  PROC DrawPart130()
    MoveL Offs(pOrigin,337.86,23.80,0.00),v40,fine,tPen\WObj:=wPaper;
    MoveL Offs(pOrigin,337.86,23.80,6.00),v60,z5,tPen\WObj:=wPaper;
    MoveL Offs(pOrigin,338.99,27.95,6.00),vTravel,z5,tPen\WObj:=wPaper;
    MoveL Offs(pOrigin,338.99,27.95,0.00),v60,z0,tPen\WObj:=wPaper;
    MoveL Offs(pOrigin,338.99,29.01,0.00),v40,fine,tPen\WObj:=wPaper;
    MoveL Offs(pOrigin,338.99,29.01,6.00),v60,z5,tPen\WObj:=wPaper;
    MoveL Offs(pOrigin,338.73,31.88,6.00),vTravel,z5,tPen\WObj:=wPaper;
    MoveL Offs(pOrigin,338.73,31.88,0.00),v60,z0,tPen\WObj:=wPaper;
    MoveL Offs(pOrigin,336.63,33.99,0.00),v40,fine,tPen\WObj:=wPaper;
    MoveL Offs(pOrigin,336.63,33.99,6.00),v60,z5,tPen\WObj:=wPaper;
    MoveL Offs(pOrigin,334.79,36.45,6.00),vTravel,z5,tPen\WObj:=wPaper;
    MoveL Offs(pOrigin,334.79,36.45,0.00),v60,z0,tPen\WObj:=wPaper;
    MoveL Offs(pOrigin,334.36,34.11,0.00),v40,z0,tPen\WObj:=wPaper;
    MoveL Offs(pOrigin,334.36,32.62,0.00),v40,z0,tPen\WObj:=wPaper;
    MoveL Offs(pOrigin,334.79,31.14,0.00),v40,fine,tPen\WObj:=wPaper;
    MoveL Offs(pOrigin,334.79,31.14,6.00),v60,z5,tPen\WObj:=wPaper;
    MoveL Offs(pOrigin,330.05,28.61,6.00),vTravel,z5,tPen\WObj:=wPaper;
    MoveL Offs(pOrigin,330.05,28.61,0.00),v60,z0,tPen\WObj:=wPaper;
    MoveL Offs(pOrigin,332.76,25.91,0.00),v40,fine,tPen\WObj:=wPaper;
    MoveL Offs(pOrigin,332.76,25.91,6.00),v60,z5,tPen\WObj:=wPaper;
    MoveL Offs(pOrigin,324.97,24.73,6.00),vTravel,z5,tPen\WObj:=wPaper;
    MoveL Offs(pOrigin,324.97,24.73,0.00),v60,z0,tPen\WObj:=wPaper;
    MoveL Offs(pOrigin,317.76,31.95,0.00),v40,z0,tPen\WObj:=wPaper;
    MoveL Offs(pOrigin,318.38,31.94,0.00),v40,z0,tPen\WObj:=wPaper;
    MoveL Offs(pOrigin,312.97,26.53,0.00),v40,z0,tPen\WObj:=wPaper;
    MoveL Offs(pOrigin,313.75,26.62,0.00),v40,z0,tPen\WObj:=wPaper;
    MoveL Offs(pOrigin,319.49,26.62,0.00),v40,fine,tPen\WObj:=wPaper;
    MoveL Offs(pOrigin,319.49,26.62,6.00),v60,z5,tPen\WObj:=wPaper;
    MoveL Offs(pOrigin,320.12,27.67,6.00),vTravel,z5,tPen\WObj:=wPaper;
    MoveL Offs(pOrigin,320.12,27.67,0.00),v60,z0,tPen\WObj:=wPaper;
    MoveL Offs(pOrigin,310.99,27.67,0.00),v40,z0,tPen\WObj:=wPaper;
    MoveL Offs(pOrigin,310.58,28.67,0.00),v40,z0,tPen\WObj:=wPaper;
    MoveL Offs(pOrigin,314.04,25.22,0.00),v40,z0,tPen\WObj:=wPaper;
    MoveL Offs(pOrigin,314.02,26.08,0.00),v40,z0,tPen\WObj:=wPaper;
    MoveL Offs(pOrigin,324.54,36.60,0.00),v40,z0,tPen\WObj:=wPaper;
    MoveL Offs(pOrigin,325.24,36.42,0.00),v40,z0,tPen\WObj:=wPaper;
    MoveL Offs(pOrigin,321.93,39.72,0.00),v40,z0,tPen\WObj:=wPaper;
    MoveL Offs(pOrigin,322.75,39.29,0.00),v40,z0,tPen\WObj:=wPaper;
    MoveL Offs(pOrigin,324.85,41.40,0.00),v40,z0,tPen\WObj:=wPaper;
    MoveL Offs(pOrigin,325.67,41.96,0.00),v40,z0,tPen\WObj:=wPaper;
    MoveL Offs(pOrigin,321.31,46.32,0.00),v40,z0,tPen\WObj:=wPaper;
    MoveL Offs(pOrigin,322.17,46.18,0.00),v40,z0,tPen\WObj:=wPaper;
    MoveL Offs(pOrigin,324.27,48.29,0.00),v40,fine,tPen\WObj:=wPaper;
    MoveL Offs(pOrigin,324.27,48.29,6.00),v60,z5,tPen\WObj:=wPaper;
    MoveL Offs(pOrigin,324.57,47.09,6.00),vTravel,z5,tPen\WObj:=wPaper;
    MoveL Offs(pOrigin,324.57,47.09,0.00),v60,z0,tPen\WObj:=wPaper;
    MoveL Offs(pOrigin,322.47,44.98,0.00),v40,z0,tPen\WObj:=wPaper;
    MoveL Offs(pOrigin,323.10,45.62,0.00),v40,z0,tPen\WObj:=wPaper;
    MoveL Offs(pOrigin,324.16,45.62,0.00),v40,z0,tPen\WObj:=wPaper;
    MoveL Offs(pOrigin,324.72,45.74,0.00),v40,z0,tPen\WObj:=wPaper;
    MoveL Offs(pOrigin,322.76,43.79,0.00),v40,z0,tPen\WObj:=wPaper;
    MoveL Offs(pOrigin,321.77,44.37,0.00),v40,z0,tPen\WObj:=wPaper;
    MoveL Offs(pOrigin,325.67,40.46,0.00),v40,z0,tPen\WObj:=wPaper;
    MoveL Offs(pOrigin,324.85,39.90,0.00),v40,z0,tPen\WObj:=wPaper;
    MoveL Offs(pOrigin,322.29,37.34,0.00),v40,z0,tPen\WObj:=wPaper;
    MoveL Offs(pOrigin,321.79,36.88,0.00),v40,z0,tPen\WObj:=wPaper;
    MoveL Offs(pOrigin,324.65,34.02,0.00),v40,z0,tPen\WObj:=wPaper;
    MoveL Offs(pOrigin,324.08,34.65,0.00),v40,z0,tPen\WObj:=wPaper;
    MoveL Offs(pOrigin,315.22,25.79,0.00),v40,z0,tPen\WObj:=wPaper;
    MoveL Offs(pOrigin,316.26,25.34,0.00),v40,z0,tPen\WObj:=wPaper;
    MoveL Offs(pOrigin,323.78,32.85,0.00),v40,z0,tPen\WObj:=wPaper;
    MoveL Offs(pOrigin,323.31,32.95,0.00),v40,z0,tPen\WObj:=wPaper;
    MoveL Offs(pOrigin,321.19,32.95,0.00),v40,z0,tPen\WObj:=wPaper;
    MoveL Offs(pOrigin,321.04,32.41,0.00),v40,z0,tPen\WObj:=wPaper;
    MoveL Offs(pOrigin,321.04,31.14,0.00),v40,z0,tPen\WObj:=wPaper;
    MoveL Offs(pOrigin,322.09,31.56,0.00),v40,z0,tPen\WObj:=wPaper;
    MoveL Offs(pOrigin,322.09,33.69,0.00),v40,z0,tPen\WObj:=wPaper;
    MoveL Offs(pOrigin,322.04,34.01,0.00),v40,z0,tPen\WObj:=wPaper;
    MoveL Offs(pOrigin,323.52,34.01,0.00),v40,z0,tPen\WObj:=wPaper;
    MoveL Offs(pOrigin,323.74,35.06,0.00),v40,z0,tPen\WObj:=wPaper;
    MoveL Offs(pOrigin,322.46,35.06,0.00),v40,z0,tPen\WObj:=wPaper;
    MoveL Offs(pOrigin,321.39,34.94,0.00),v40,z0,tPen\WObj:=wPaper;
    MoveL Offs(pOrigin,324.69,38.25,0.00),v40,z0,tPen\WObj:=wPaper;
    MoveL Offs(pOrigin,325.38,37.76,0.00),v40,z0,tPen\WObj:=wPaper;
    MoveL Offs(pOrigin,321.93,41.22,0.00),v40,fine,tPen\WObj:=wPaper;
    MoveL Offs(pOrigin,321.93,41.22,6.00),v60,z5,tPen\WObj:=wPaper;
    MoveL Offs(pOrigin,321.92,42.72,6.00),vTravel,z5,tPen\WObj:=wPaper;
    MoveL Offs(pOrigin,321.92,42.72,0.00),v60,z0,tPen\WObj:=wPaper;
    MoveL Offs(pOrigin,325.38,39.26,0.00),v40,fine,tPen\WObj:=wPaper;
    MoveL Offs(pOrigin,325.38,39.26,6.00),v60,z5,tPen\WObj:=wPaper;
    MoveL Offs(pOrigin,323.95,36.12,6.00),vTravel,z5,tPen\WObj:=wPaper;
    MoveL Offs(pOrigin,323.95,36.12,0.00),v60,z0,tPen\WObj:=wPaper;
    MoveL Offs(pOrigin,322.89,36.12,0.00),v40,z0,tPen\WObj:=wPaper;
    MoveL Offs(pOrigin,322.46,36.24,0.00),v40,z0,tPen\WObj:=wPaper;
    MoveL Offs(pOrigin,322.25,34.75,0.00),v40,z0,tPen\WObj:=wPaper;
    MoveL Offs(pOrigin,321.40,34.33,0.00),v40,z0,tPen\WObj:=wPaper;
    MoveL Offs(pOrigin,320.90,34.78,0.00),v40,z0,tPen\WObj:=wPaper;
    MoveL Offs(pOrigin,323.90,31.78,0.00),v40,z0,tPen\WObj:=wPaper;
    MoveL Offs(pOrigin,322.89,31.90,0.00),v40,z0,tPen\WObj:=wPaper;
    MoveL Offs(pOrigin,319.91,31.90,0.00),v40,fine,tPen\WObj:=wPaper;
    MoveL Offs(pOrigin,319.91,31.90,6.00),v60,z5,tPen\WObj:=wPaper;
    MoveL Offs(pOrigin,318.81,32.39,6.00),vTravel,z5,tPen\WObj:=wPaper;
    MoveL Offs(pOrigin,318.81,32.39,0.00),v60,z0,tPen\WObj:=wPaper;
    MoveL Offs(pOrigin,322.41,28.79,0.00),v40,z0,tPen\WObj:=wPaper;
    MoveL Offs(pOrigin,322.04,29.23,0.00),v40,z0,tPen\WObj:=wPaper;
    MoveL Offs(pOrigin,322.25,29.65,0.00),v40,z0,tPen\WObj:=wPaper;
    MoveL Offs(pOrigin,322.04,29.23,0.00),v40,z0,tPen\WObj:=wPaper;
    MoveL Offs(pOrigin,321.82,29.78,0.00),v40,z0,tPen\WObj:=wPaper;
    MoveL Offs(pOrigin,320.76,29.78,0.00),v40,fine,tPen\WObj:=wPaper;
    MoveL Offs(pOrigin,320.76,29.78,6.00),v60,z5,tPen\WObj:=wPaper;
    MoveL Offs(pOrigin,319.70,28.80,6.00),vTravel,z5,tPen\WObj:=wPaper;
    MoveL Offs(pOrigin,319.70,28.80,0.00),v60,z0,tPen\WObj:=wPaper;
    MoveL Offs(pOrigin,320.55,29.65,0.00),v40,z0,tPen\WObj:=wPaper;
    MoveL Offs(pOrigin,319.70,28.80,0.00),v40,fine,tPen\WObj:=wPaper;
    MoveL Offs(pOrigin,319.70,28.80,6.00),v60,z5,tPen\WObj:=wPaper;
    MoveL Offs(pOrigin,321.19,28.16,6.00),vTravel,z5,tPen\WObj:=wPaper;
    MoveL Offs(pOrigin,321.19,28.16,0.00),v60,z0,tPen\WObj:=wPaper;
    MoveL Offs(pOrigin,321.61,28.59,0.00),v40,z0,tPen\WObj:=wPaper;
    MoveL Offs(pOrigin,321.19,28.16,0.00),v40,z0,tPen\WObj:=wPaper;
    MoveL Offs(pOrigin,321.06,27.15,0.00),v40,z0,tPen\WObj:=wPaper;
    MoveL Offs(pOrigin,318.66,24.75,0.00),v40,z0,tPen\WObj:=wPaper;
    MoveL Offs(pOrigin,318.23,24.01,0.00),v40,z0,tPen\WObj:=wPaper;
    MoveL Offs(pOrigin,312.37,29.87,0.00),v40,z0,tPen\WObj:=wPaper;
    MoveL Offs(pOrigin,313.12,30.61,0.00),v40,z0,tPen\WObj:=wPaper;
    MoveL Offs(pOrigin,319.73,24.00,0.00),v40,z0,tPen\WObj:=wPaper;
    MoveL Offs(pOrigin,320.16,24.75,0.00),v40,z0,tPen\WObj:=wPaper;
    MoveL Offs(pOrigin,322.41,27.01,0.00),v40,fine,tPen\WObj:=wPaper;
    MoveL Offs(pOrigin,322.41,27.01,6.00),v60,z5,tPen\WObj:=wPaper;
    MoveL Offs(pOrigin,324.16,25.56,6.00),vTravel,z5,tPen\WObj:=wPaper;
    MoveL Offs(pOrigin,324.16,25.56,0.00),v60,z0,tPen\WObj:=wPaper;
  ENDPROC

  PROC DrawPart131()
    MoveL Offs(pOrigin,316.73,25.56,0.00),v40,z0,tPen\WObj:=wPaper;
    MoveL Offs(pOrigin,316.81,26.04,0.00),v40,z0,tPen\WObj:=wPaper;
    MoveL Offs(pOrigin,316.81,27.10,0.00),v40,fine,tPen\WObj:=wPaper;
    MoveL Offs(pOrigin,316.81,27.10,6.00),v60,z5,tPen\WObj:=wPaper;
    MoveL Offs(pOrigin,315.45,28.16,6.00),vTravel,z5,tPen\WObj:=wPaper;
    MoveL Offs(pOrigin,315.45,28.16,0.00),v60,z0,tPen\WObj:=wPaper;
    MoveL Offs(pOrigin,318.00,27.95,0.00),v40,z0,tPen\WObj:=wPaper;
    MoveL Offs(pOrigin,319.06,28.30,0.00),v40,z0,tPen\WObj:=wPaper;
    MoveL Offs(pOrigin,320.55,29.44,0.00),v40,z0,tPen\WObj:=wPaper;
    MoveL Offs(pOrigin,320.76,30.50,0.00),v40,z0,tPen\WObj:=wPaper;
    MoveL Offs(pOrigin,320.55,30.71,0.00),v40,z0,tPen\WObj:=wPaper;
    MoveL Offs(pOrigin,315.88,28.94,0.00),v40,z0,tPen\WObj:=wPaper;
    MoveL Offs(pOrigin,315.02,28.16,0.00),v40,z0,tPen\WObj:=wPaper;
    MoveL Offs(pOrigin,314.70,28.59,0.00),v40,z0,tPen\WObj:=wPaper;
    MoveL Offs(pOrigin,314.70,26.89,0.00),v40,z0,tPen\WObj:=wPaper;
    MoveL Offs(pOrigin,313.65,27.10,0.00),v40,z0,tPen\WObj:=wPaper;
    MoveL Offs(pOrigin,313.65,28.59,0.00),v40,z0,tPen\WObj:=wPaper;
    MoveL Offs(pOrigin,313.11,28.73,0.00),v40,z0,tPen\WObj:=wPaper;
    MoveL Offs(pOrigin,315.88,28.73,0.00),v40,z0,tPen\WObj:=wPaper;
    MoveL Offs(pOrigin,315.45,29.78,0.00),v40,z0,tPen\WObj:=wPaper;
    MoveL Offs(pOrigin,317.79,29.78,0.00),v40,z0,tPen\WObj:=wPaper;
    MoveL Offs(pOrigin,318.00,30.84,0.00),v40,z0,tPen\WObj:=wPaper;
    MoveL Offs(pOrigin,322.46,30.84,0.00),v40,z0,tPen\WObj:=wPaper;
    MoveL Offs(pOrigin,322.87,30.46,0.00),v40,z0,tPen\WObj:=wPaper;
    MoveL Offs(pOrigin,317.31,24.90,0.00),v40,z0,tPen\WObj:=wPaper;
    MoveL Offs(pOrigin,316.29,24.46,0.00),v40,z0,tPen\WObj:=wPaper;
    MoveL Offs(pOrigin,311.48,29.27,0.00),v40,fine,tPen\WObj:=wPaper;
    MoveL Offs(pOrigin,311.48,29.27,6.00),v60,z5,tPen\WObj:=wPaper;
    MoveL Offs(pOrigin,313.75,29.65,6.00),vTravel,z5,tPen\WObj:=wPaper;
    MoveL Offs(pOrigin,313.75,29.65,0.00),v60,z0,tPen\WObj:=wPaper;
    MoveL Offs(pOrigin,309.92,27.45,0.00),v40,z0,tPen\WObj:=wPaper;
    MoveL Offs(pOrigin,305.89,26.25,0.00),v40,z0,tPen\WObj:=wPaper;
    MoveL Offs(pOrigin,303.12,25.83,0.00),v40,z0,tPen\WObj:=wPaper;
    MoveL Offs(pOrigin,297.60,25.83,0.00),v40,z0,tPen\WObj:=wPaper;
    MoveL Offs(pOrigin,295.69,26.25,0.00),v40,z0,tPen\WObj:=wPaper;
    MoveL Offs(pOrigin,296.11,27.45,0.00),v40,z0,tPen\WObj:=wPaper;
    MoveL Offs(pOrigin,297.60,27.95,0.00),v40,z0,tPen\WObj:=wPaper;
    MoveL Offs(pOrigin,297.60,27.95,0.00),v40,z0,tPen\WObj:=wPaper;
    MoveL Offs(pOrigin,298.52,29.37,0.00),v40,z0,tPen\WObj:=wPaper;
    MoveL Offs(pOrigin,299.73,29.30,0.00),v40,z0,tPen\WObj:=wPaper;
    MoveL Offs(pOrigin,301.42,30.71,0.00),v40,fine,tPen\WObj:=wPaper;
    MoveL Offs(pOrigin,301.42,30.71,6.00),v60,z5,tPen\WObj:=wPaper;
    MoveL Offs(pOrigin,303.40,26.90,6.00),vTravel,z5,tPen\WObj:=wPaper;
    MoveL Offs(pOrigin,303.40,26.90,0.00),v60,z0,tPen\WObj:=wPaper;
    MoveL Offs(pOrigin,306.25,24.04,0.00),v40,fine,tPen\WObj:=wPaper;
    MoveL Offs(pOrigin,306.25,24.04,6.00),v60,z5,tPen\WObj:=wPaper;
    MoveL Offs(pOrigin,307.59,25.56,6.00),vTravel,z5,tPen\WObj:=wPaper;
    MoveL Offs(pOrigin,307.59,25.56,0.00),v60,z0,tPen\WObj:=wPaper;
    MoveL Offs(pOrigin,302.27,25.56,0.00),v40,fine,tPen\WObj:=wPaper;
    MoveL Offs(pOrigin,302.27,25.56,6.00),v60,z5,tPen\WObj:=wPaper;
    MoveL Offs(pOrigin,298.15,27.66,6.00),vTravel,z5,tPen\WObj:=wPaper;
    MoveL Offs(pOrigin,298.15,27.66,0.00),v60,z0,tPen\WObj:=wPaper;
    MoveL Offs(pOrigin,297.10,28.71,0.00),v40,fine,tPen\WObj:=wPaper;
    MoveL Offs(pOrigin,297.10,28.71,6.00),v60,z5,tPen\WObj:=wPaper;
    MoveL Offs(pOrigin,296.64,26.63,6.00),vTravel,z5,tPen\WObj:=wPaper;
    MoveL Offs(pOrigin,296.64,26.63,0.00),v60,z0,tPen\WObj:=wPaper;
    MoveL Offs(pOrigin,294.69,24.68,0.00),v40,z0,tPen\WObj:=wPaper;
    MoveL Offs(pOrigin,294.27,24.08,0.00),v40,z0,tPen\WObj:=wPaper;
    MoveL Offs(pOrigin,291.41,26.93,0.00),v40,fine,tPen\WObj:=wPaper;
    MoveL Offs(pOrigin,291.41,26.93,6.00),v60,z5,tPen\WObj:=wPaper;
    MoveL Offs(pOrigin,309.22,25.77,6.00),vTravel,z5,tPen\WObj:=wPaper;
    MoveL Offs(pOrigin,309.22,25.77,0.00),v60,z0,tPen\WObj:=wPaper;
    MoveL Offs(pOrigin,313.73,30.28,0.00),v40,fine,tPen\WObj:=wPaper;
    MoveL Offs(pOrigin,313.73,30.28,6.00),v60,z5,tPen\WObj:=wPaper;
    MoveL Offs(pOrigin,313.72,31.51,6.00),vTravel,z5,tPen\WObj:=wPaper;
    MoveL Offs(pOrigin,313.72,31.51,0.00),v60,z0,tPen\WObj:=wPaper;
    MoveL Offs(pOrigin,321.08,24.15,0.00),v40,fine,tPen\WObj:=wPaper;
    MoveL Offs(pOrigin,321.08,24.15,6.00),v60,z5,tPen\WObj:=wPaper;
    MoveL Offs(pOrigin,323.16,29.53,6.00),vTravel,z5,tPen\WObj:=wPaper;
    MoveL Offs(pOrigin,323.16,29.53,0.00),v60,z0,tPen\WObj:=wPaper;
    MoveL Offs(pOrigin,319.55,33.14,0.00),v40,z0,tPen\WObj:=wPaper;
    MoveL Offs(pOrigin,320.30,33.89,0.00),v40,z0,tPen\WObj:=wPaper;
    MoveL Offs(pOrigin,323.46,30.73,0.00),v40,fine,tPen\WObj:=wPaper;
    MoveL Offs(pOrigin,323.46,30.73,6.00),v60,z5,tPen\WObj:=wPaper;
    MoveL Offs(pOrigin,324.35,32.82,6.00),vTravel,z5,tPen\WObj:=wPaper;
    MoveL Offs(pOrigin,324.35,32.82,0.00),v60,z0,tPen\WObj:=wPaper;
    MoveL Offs(pOrigin,321.34,35.83,0.00),v40,fine,tPen\WObj:=wPaper;
    MoveL Offs(pOrigin,321.34,35.83,6.00),v60,z5,tPen\WObj:=wPaper;
    MoveL Offs(pOrigin,321.94,38.22,6.00),vTravel,z5,tPen\WObj:=wPaper;
    MoveL Offs(pOrigin,321.94,38.22,0.00),v60,z0,tPen\WObj:=wPaper;
    MoveL Offs(pOrigin,324.79,35.37,0.00),v40,fine,tPen\WObj:=wPaper;
    MoveL Offs(pOrigin,324.79,35.37,6.00),v60,z5,tPen\WObj:=wPaper;
    MoveL Offs(pOrigin,325.21,46.90,6.00),vTravel,z5,tPen\WObj:=wPaper;
    MoveL Offs(pOrigin,325.21,46.90,0.00),v60,z0,tPen\WObj:=wPaper;
    MoveL Offs(pOrigin,317.84,54.27,0.00),v40,fine,tPen\WObj:=wPaper;
    MoveL Offs(pOrigin,317.84,54.27,6.00),v60,z5,tPen\WObj:=wPaper;
    MoveL Offs(pOrigin,321.61,51.96,6.00),vTravel,z5,tPen\WObj:=wPaper;
    MoveL Offs(pOrigin,321.61,51.96,0.00),v60,z0,tPen\WObj:=wPaper;
    MoveL Offs(pOrigin,322.68,51.96,0.00),v40,z0,tPen\WObj:=wPaper;
    MoveL Offs(pOrigin,323.24,51.73,0.00),v40,z0,tPen\WObj:=wPaper;
    MoveL Offs(pOrigin,321.43,49.92,0.00),v40,fine,tPen\WObj:=wPaper;
    MoveL Offs(pOrigin,321.43,49.92,6.00),v60,z5,tPen\WObj:=wPaper;
    MoveL Offs(pOrigin,336.12,53.91,6.00),vTravel,z5,tPen\WObj:=wPaper;
    MoveL Offs(pOrigin,336.12,53.91,0.00),v60,z0,tPen\WObj:=wPaper;
    MoveL Offs(pOrigin,338.37,51.66,0.00),v40,fine,tPen\WObj:=wPaper;
    MoveL Offs(pOrigin,338.37,51.66,6.00),v60,z5,tPen\WObj:=wPaper;
    MoveL Offs(pOrigin,341.22,53.28,6.00),vTravel,z5,tPen\WObj:=wPaper;
    MoveL Offs(pOrigin,341.22,53.28,0.00),v60,z0,tPen\WObj:=wPaper;
    MoveL Offs(pOrigin,342.72,54.78,0.00),v40,z0,tPen\WObj:=wPaper;
    MoveL Offs(pOrigin,342.23,54.94,0.00),v40,z0,tPen\WObj:=wPaper;
    MoveL Offs(pOrigin,341.59,55.58,0.00),v40,z0,tPen\WObj:=wPaper;
    MoveL Offs(pOrigin,342.23,54.94,0.00),v40,fine,tPen\WObj:=wPaper;
    MoveL Offs(pOrigin,342.23,54.94,6.00),v60,z5,tPen\WObj:=wPaper;
    MoveL Offs(pOrigin,341.59,53.24,6.00),vTravel,z5,tPen\WObj:=wPaper;
    MoveL Offs(pOrigin,341.59,53.24,0.00),v60,z0,tPen\WObj:=wPaper;
    MoveL Offs(pOrigin,340.95,54.09,0.00),v40,z0,tPen\WObj:=wPaper;
    MoveL Offs(pOrigin,341.59,53.24,0.00),v40,fine,tPen\WObj:=wPaper;
    MoveL Offs(pOrigin,341.59,53.24,6.00),v60,z5,tPen\WObj:=wPaper;
    MoveL Offs(pOrigin,342.86,51.96,6.00),vTravel,z5,tPen\WObj:=wPaper;
    MoveL Offs(pOrigin,342.86,51.96,0.00),v60,z0,tPen\WObj:=wPaper;
    MoveL Offs(pOrigin,344.14,51.96,0.00),v40,z0,tPen\WObj:=wPaper;
    MoveL Offs(pOrigin,344.14,52.17,0.00),v40,z0,tPen\WObj:=wPaper;
    MoveL Offs(pOrigin,343.71,52.81,0.00),v40,z0,tPen\WObj:=wPaper;
    MoveL Offs(pOrigin,344.14,52.17,0.00),v40,z0,tPen\WObj:=wPaper;
    MoveL Offs(pOrigin,344.66,52.24,0.00),v40,z0,tPen\WObj:=wPaper;
    MoveL Offs(pOrigin,343.01,50.59,0.00),v40,z0,tPen\WObj:=wPaper;
    MoveL Offs(pOrigin,343.50,50.90,0.00),v40,z0,tPen\WObj:=wPaper;
    MoveL Offs(pOrigin,344.78,50.90,0.00),v40,fine,tPen\WObj:=wPaper;
    MoveL Offs(pOrigin,344.78,50.90,6.00),v60,z5,tPen\WObj:=wPaper;
    MoveL Offs(pOrigin,343.71,50.26,6.00),vTravel,z5,tPen\WObj:=wPaper;
  ENDPROC

  PROC DrawPart132()
    MoveL Offs(pOrigin,343.71,50.26,0.00),v60,z0,tPen\WObj:=wPaper;
    MoveL Offs(pOrigin,343.29,50.90,0.00),v40,z0,tPen\WObj:=wPaper;
    MoveL Offs(pOrigin,343.71,50.26,0.00),v40,fine,tPen\WObj:=wPaper;
    MoveL Offs(pOrigin,343.71,50.26,6.00),v60,z5,tPen\WObj:=wPaper;
    MoveL Offs(pOrigin,346.90,45.62,6.00),vTravel,z5,tPen\WObj:=wPaper;
    MoveL Offs(pOrigin,346.90,45.62,0.00),v60,z0,tPen\WObj:=wPaper;
    MoveL Offs(pOrigin,347.96,45.62,0.00),v40,fine,tPen\WObj:=wPaper;
    MoveL Offs(pOrigin,347.96,45.62,6.00),v60,z5,tPen\WObj:=wPaper;
    MoveL Offs(pOrigin,346.69,45.38,6.00),vTravel,z5,tPen\WObj:=wPaper;
    MoveL Offs(pOrigin,346.69,45.38,0.00),v60,z0,tPen\WObj:=wPaper;
    MoveL Offs(pOrigin,346.26,46.01,0.00),v40,z0,tPen\WObj:=wPaper;
    MoveL Offs(pOrigin,346.69,45.38,0.00),v40,fine,tPen\WObj:=wPaper;
    MoveL Offs(pOrigin,346.69,45.38,6.00),v60,z5,tPen\WObj:=wPaper;
    MoveL Offs(pOrigin,344.14,26.67,6.00),vTravel,z5,tPen\WObj:=wPaper;
    MoveL Offs(pOrigin,344.14,26.67,0.00),v60,z0,tPen\WObj:=wPaper;
    MoveL Offs(pOrigin,344.77,27.10,0.00),v40,z0,tPen\WObj:=wPaper;
    MoveL Offs(pOrigin,344.14,26.67,0.00),v40,fine,tPen\WObj:=wPaper;
    MoveL Offs(pOrigin,344.14,26.67,6.00),v60,z5,tPen\WObj:=wPaper;
    MoveL Offs(pOrigin,303.76,40.06,6.00),vTravel,z5,tPen\WObj:=wPaper;
    MoveL Offs(pOrigin,303.76,40.06,0.00),v60,z0,tPen\WObj:=wPaper;
    MoveL Offs(pOrigin,302.70,45.59,0.00),v40,z0,tPen\WObj:=wPaper;
    MoveL Offs(pOrigin,301.42,49.41,0.00),v40,fine,tPen\WObj:=wPaper;
    MoveL Offs(pOrigin,301.42,49.41,6.00),v60,z5,tPen\WObj:=wPaper;
    MoveL Offs(pOrigin,296.75,57.28,6.00),vTravel,z5,tPen\WObj:=wPaper;
    MoveL Offs(pOrigin,296.75,57.28,0.00),v60,z0,tPen\WObj:=wPaper;
    MoveL Offs(pOrigin,292.50,61.53,0.00),v40,fine,tPen\WObj:=wPaper;
    MoveL Offs(pOrigin,292.50,61.53,6.00),v60,z5,tPen\WObj:=wPaper;
    MoveL Offs(pOrigin,294.60,61.08,6.00),vTravel,z5,tPen\WObj:=wPaper;
    MoveL Offs(pOrigin,294.60,61.08,0.00),v60,z0,tPen\WObj:=wPaper;
    MoveL Offs(pOrigin,284.38,71.30,0.00),v40,z0,tPen\WObj:=wPaper;
    MoveL Offs(pOrigin,284.95,71.68,0.00),v40,z0,tPen\WObj:=wPaper;
    MoveL Offs(pOrigin,287.65,74.39,0.00),v40,z0,tPen\WObj:=wPaper;
    MoveL Offs(pOrigin,286.98,74.14,0.00),v40,z0,tPen\WObj:=wPaper;
    MoveL Offs(pOrigin,285.91,74.14,0.00),v40,z0,tPen\WObj:=wPaper;
    MoveL Offs(pOrigin,285.25,73.48,0.00),v40,z0,tPen\WObj:=wPaper;
    MoveL Offs(pOrigin,287.81,76.04,0.00),v40,z0,tPen\WObj:=wPaper;
    MoveL Offs(pOrigin,287.40,76.25,0.00),v40,z0,tPen\WObj:=wPaper;
    MoveL Offs(pOrigin,286.34,76.25,0.00),v40,z0,tPen\WObj:=wPaper;
    MoveL Offs(pOrigin,285.56,76.78,0.00),v40,z0,tPen\WObj:=wPaper;
    MoveL Offs(pOrigin,288.42,79.63,0.00),v40,z0,tPen\WObj:=wPaper;
    MoveL Offs(pOrigin,288.04,79.42,0.00),v40,z0,tPen\WObj:=wPaper;
    MoveL Offs(pOrigin,286.76,79.42,0.00),v40,z0,tPen\WObj:=wPaper;
    MoveL Offs(pOrigin,286.02,78.73,0.00),v40,z0,tPen\WObj:=wPaper;
    MoveL Offs(pOrigin,288.87,81.58,0.00),v40,z0,tPen\WObj:=wPaper;
    MoveL Offs(pOrigin,288.46,81.53,0.00),v40,z0,tPen\WObj:=wPaper;
    MoveL Offs(pOrigin,287.19,81.53,0.00),v40,z0,tPen\WObj:=wPaper;
    MoveL Offs(pOrigin,286.63,82.32,0.00),v40,z0,tPen\WObj:=wPaper;
    MoveL Offs(pOrigin,289.78,85.48,0.00),v40,z0,tPen\WObj:=wPaper;
    MoveL Offs(pOrigin,289.31,85.75,0.00),v40,z0,tPen\WObj:=wPaper;
    MoveL Offs(pOrigin,288.04,85.75,0.00),v40,z0,tPen\WObj:=wPaper;
    MoveL Offs(pOrigin,287.54,86.22,0.00),v40,z0,tPen\WObj:=wPaper;
    MoveL Offs(pOrigin,292.35,91.03,0.00),v40,z0,tPen\WObj:=wPaper;
    MoveL Offs(pOrigin,293.01,91.04,0.00),v40,z0,tPen\WObj:=wPaper;
    MoveL Offs(pOrigin,289.11,94.95,0.00),v40,fine,tPen\WObj:=wPaper;
    MoveL Offs(pOrigin,289.11,94.95,6.00),v60,z5,tPen\WObj:=wPaper;
    MoveL Offs(pOrigin,289.40,96.15,6.00),vTravel,z5,tPen\WObj:=wPaper;
    MoveL Offs(pOrigin,289.40,96.15,0.00),v60,z0,tPen\WObj:=wPaper;
    MoveL Offs(pOrigin,293.01,92.54,0.00),v40,z0,tPen\WObj:=wPaper;
    MoveL Offs(pOrigin,292.35,92.53,0.00),v40,z0,tPen\WObj:=wPaper;
    MoveL Offs(pOrigin,287.99,88.17,0.00),v40,z0,tPen\WObj:=wPaper;
    MoveL Offs(pOrigin,288.46,87.86,0.00),v40,z0,tPen\WObj:=wPaper;
    MoveL Offs(pOrigin,289.74,87.86,0.00),v40,z0,tPen\WObj:=wPaper;
    MoveL Offs(pOrigin,290.09,87.28,0.00),v40,z0,tPen\WObj:=wPaper;
    MoveL Offs(pOrigin,287.08,84.27,0.00),v40,z0,tPen\WObj:=wPaper;
    MoveL Offs(pOrigin,286.59,84.02,0.00),v40,z0,tPen\WObj:=wPaper;
    MoveL Offs(pOrigin,289.30,81.32,0.00),v40,fine,tPen\WObj:=wPaper;
    MoveL Offs(pOrigin,289.30,81.32,6.00),v60,z5,tPen\WObj:=wPaper;
    MoveL Offs(pOrigin,289.00,80.12,6.00),vTravel,z5,tPen\WObj:=wPaper;
    MoveL Offs(pOrigin,289.00,80.12,0.00),v60,z0,tPen\WObj:=wPaper;
    MoveL Offs(pOrigin,286.30,82.82,0.00),v40,z0,tPen\WObj:=wPaper;
    MoveL Offs(pOrigin,287.40,82.58,0.00),v40,z0,tPen\WObj:=wPaper;
    MoveL Offs(pOrigin,288.68,82.58,0.00),v40,z0,tPen\WObj:=wPaper;
    MoveL Offs(pOrigin,289.59,82.51,0.00),v40,z0,tPen\WObj:=wPaper;
    MoveL Offs(pOrigin,286.89,85.22,0.00),v40,z0,tPen\WObj:=wPaper;
    MoveL Offs(pOrigin,287.82,84.70,0.00),v40,z0,tPen\WObj:=wPaper;
    MoveL Offs(pOrigin,289.10,84.70,0.00),v40,z0,tPen\WObj:=wPaper;
    MoveL Offs(pOrigin,288.89,83.64,0.00),v40,z0,tPen\WObj:=wPaper;
    MoveL Offs(pOrigin,287.61,83.64,0.00),v40,fine,tPen\WObj:=wPaper;
    MoveL Offs(pOrigin,287.61,83.64,6.00),v60,z5,tPen\WObj:=wPaper;
    MoveL Offs(pOrigin,289.33,83.53,6.00),vTravel,z5,tPen\WObj:=wPaper;
    MoveL Offs(pOrigin,289.33,83.53,0.00),v60,z0,tPen\WObj:=wPaper;
    MoveL Offs(pOrigin,286.32,80.53,0.00),v40,z0,tPen\WObj:=wPaper;
    MoveL Offs(pOrigin,285.86,80.28,0.00),v40,z0,tPen\WObj:=wPaper;
    MoveL Offs(pOrigin,288.71,77.42,0.00),v40,z0,tPen\WObj:=wPaper;
    MoveL Offs(pOrigin,288.26,77.99,0.00),v40,z0,tPen\WObj:=wPaper;
    MoveL Offs(pOrigin,285.41,75.13,0.00),v40,z0,tPen\WObj:=wPaper;
    MoveL Offs(pOrigin,284.97,75.19,0.00),v40,z0,tPen\WObj:=wPaper;
    MoveL Offs(pOrigin,287.83,72.33,0.00),v40,z0,tPen\WObj:=wPaper;
    MoveL Offs(pOrigin,287.35,72.59,0.00),v40,z0,tPen\WObj:=wPaper;
    MoveL Offs(pOrigin,281.49,66.73,0.00),v40,z0,tPen\WObj:=wPaper;
    MoveL Offs(pOrigin,282.00,66.21,0.00),v40,z0,tPen\WObj:=wPaper;
    MoveL Offs(pOrigin,279.45,68.76,0.00),v40,z0,tPen\WObj:=wPaper;
    MoveL Offs(pOrigin,280.50,69.21,0.00),v40,z0,tPen\WObj:=wPaper;
    MoveL Offs(pOrigin,283.50,66.21,0.00),v40,z0,tPen\WObj:=wPaper;
    MoveL Offs(pOrigin,283.14,66.88,0.00),v40,z0,tPen\WObj:=wPaper;
    MoveL Offs(pOrigin,287.19,70.94,0.00),v40,z0,tPen\WObj:=wPaper;
    MoveL Offs(pOrigin,287.68,70.99,0.00),v40,z0,tPen\WObj:=wPaper;
    MoveL Offs(pOrigin,284.83,73.84,0.00),v40,z0,tPen\WObj:=wPaper;
    MoveL Offs(pOrigin,285.70,73.08,0.00),v40,z0,tPen\WObj:=wPaper;
    MoveL Offs(pOrigin,286.76,73.08,0.00),v40,z0,tPen\WObj:=wPaper;
    MoveL Offs(pOrigin,286.76,72.02,0.00),v40,z0,tPen\WObj:=wPaper;
    MoveL Offs(pOrigin,285.70,72.02,0.00),v40,z0,tPen\WObj:=wPaper;
    MoveL Offs(pOrigin,285.49,70.97,0.00),v40,z0,tPen\WObj:=wPaper;
    MoveL Offs(pOrigin,286.55,70.97,0.00),v40,z0,tPen\WObj:=wPaper;
    MoveL Offs(pOrigin,286.34,69.91,0.00),v40,z0,tPen\WObj:=wPaper;
    MoveL Offs(pOrigin,285.27,69.91,0.00),v40,z0,tPen\WObj:=wPaper;
    MoveL Offs(pOrigin,284.85,68.86,0.00),v40,z0,tPen\WObj:=wPaper;
    MoveL Offs(pOrigin,286.34,68.86,0.00),v40,z0,tPen\WObj:=wPaper;
    MoveL Offs(pOrigin,286.89,69.14,0.00),v40,z0,tPen\WObj:=wPaper;
    MoveL Offs(pOrigin,284.48,66.74,0.00),v40,z0,tPen\WObj:=wPaper;
    MoveL Offs(pOrigin,285.13,67.26,0.00),v40,z0,tPen\WObj:=wPaper;
    MoveL Offs(pOrigin,285.13,68.75,0.00),v40,fine,tPen\WObj:=wPaper;
    MoveL Offs(pOrigin,285.13,68.75,6.00),v60,z5,tPen\WObj:=wPaper;
    MoveL Offs(pOrigin,287.69,69.49,6.00),vTravel,z5,tPen\WObj:=wPaper;
    MoveL Offs(pOrigin,287.69,69.49,0.00),v60,z0,tPen\WObj:=wPaper;
    MoveL Offs(pOrigin,284.53,72.64,0.00),v40,fine,tPen\WObj:=wPaper;
    MoveL Offs(pOrigin,284.53,72.64,6.00),v60,z5,tPen\WObj:=wPaper;
    MoveL Offs(pOrigin,286.12,75.19,6.00),vTravel,z5,tPen\WObj:=wPaper;
    MoveL Offs(pOrigin,286.12,75.19,0.00),v60,z0,tPen\WObj:=wPaper;
    MoveL Offs(pOrigin,287.19,75.19,0.00),v40,z0,tPen\WObj:=wPaper;
  ENDPROC

  PROC DrawPart133()
    MoveL Offs(pOrigin,288.27,74.88,0.00),v40,z0,tPen\WObj:=wPaper;
    MoveL Offs(pOrigin,285.41,77.73,0.00),v40,fine,tPen\WObj:=wPaper;
    MoveL Offs(pOrigin,285.41,77.73,6.00),v60,z5,tPen\WObj:=wPaper;
    MoveL Offs(pOrigin,286.55,77.30,6.00),vTravel,z5,tPen\WObj:=wPaper;
    MoveL Offs(pOrigin,286.55,77.30,0.00),v60,z0,tPen\WObj:=wPaper;
    MoveL Offs(pOrigin,287.61,77.30,0.00),v40,z0,tPen\WObj:=wPaper;
    MoveL Offs(pOrigin,287.82,78.36,0.00),v40,z0,tPen\WObj:=wPaper;
    MoveL Offs(pOrigin,286.55,78.36,0.00),v40,fine,tPen\WObj:=wPaper;
    MoveL Offs(pOrigin,286.55,78.36,6.00),v60,z5,tPen\WObj:=wPaper;
    MoveL Offs(pOrigin,285.56,79.08,6.00),vTravel,z5,tPen\WObj:=wPaper;
    MoveL Offs(pOrigin,285.56,79.08,0.00),v60,z0,tPen\WObj:=wPaper;
    MoveL Offs(pOrigin,288.41,76.23,0.00),v40,fine,tPen\WObj:=wPaper;
    MoveL Offs(pOrigin,288.41,76.23,6.00),v60,z5,tPen\WObj:=wPaper;
    MoveL Offs(pOrigin,288.86,78.77,6.00),vTravel,z5,tPen\WObj:=wPaper;
    MoveL Offs(pOrigin,288.86,78.77,0.00),v60,z0,tPen\WObj:=wPaper;
    MoveL Offs(pOrigin,286.00,81.63,0.00),v40,fine,tPen\WObj:=wPaper;
    MoveL Offs(pOrigin,286.00,81.63,6.00),v60,z5,tPen\WObj:=wPaper;
    MoveL Offs(pOrigin,286.98,80.47,6.00),vTravel,z5,tPen\WObj:=wPaper;
    MoveL Offs(pOrigin,286.98,80.47,0.00),v60,z0,tPen\WObj:=wPaper;
    MoveL Offs(pOrigin,288.25,80.47,0.00),v40,fine,tPen\WObj:=wPaper;
    MoveL Offs(pOrigin,288.25,80.47,6.00),v60,z5,tPen\WObj:=wPaper;
    MoveL Offs(pOrigin,290.95,81.16,6.00),vTravel,z5,tPen\WObj:=wPaper;
    MoveL Offs(pOrigin,290.95,81.16,0.00),v60,z0,tPen\WObj:=wPaper;
    MoveL Offs(pOrigin,293.35,78.76,0.00),v40,fine,tPen\WObj:=wPaper;
    MoveL Offs(pOrigin,293.35,78.76,6.00),v60,z5,tPen\WObj:=wPaper;
    MoveL Offs(pOrigin,293.35,77.26,6.00),vTravel,z5,tPen\WObj:=wPaper;
    MoveL Offs(pOrigin,293.35,77.26,0.00),v60,z0,tPen\WObj:=wPaper;
    MoveL Offs(pOrigin,290.95,79.66,0.00),v40,z0,tPen\WObj:=wPaper;
    MoveL Offs(pOrigin,291.71,79.94,0.00),v40,z0,tPen\WObj:=wPaper;
    MoveL Offs(pOrigin,292.47,80.69,0.00),v40,z0,tPen\WObj:=wPaper;
    MoveL Offs(pOrigin,293.35,80.26,0.00),v40,z0,tPen\WObj:=wPaper;
    MoveL Offs(pOrigin,290.94,82.66,0.00),v40,fine,tPen\WObj:=wPaper;
    MoveL Offs(pOrigin,290.94,82.66,6.00),v60,z5,tPen\WObj:=wPaper;
    MoveL Offs(pOrigin,289.89,83.71,6.00),vTravel,z5,tPen\WObj:=wPaper;
    MoveL Offs(pOrigin,289.89,83.71,0.00),v60,z0,tPen\WObj:=wPaper;
    MoveL Offs(pOrigin,287.03,86.57,0.00),v40,fine,tPen\WObj:=wPaper;
    MoveL Offs(pOrigin,287.03,86.57,6.00),v60,z5,tPen\WObj:=wPaper;
    MoveL Offs(pOrigin,287.33,87.76,6.00),vTravel,z5,tPen\WObj:=wPaper;
    MoveL Offs(pOrigin,287.33,87.76,0.00),v60,z0,tPen\WObj:=wPaper;
    MoveL Offs(pOrigin,293.04,82.05,0.00),v40,fine,tPen\WObj:=wPaper;
    MoveL Offs(pOrigin,293.04,82.05,6.00),v60,z5,tPen\WObj:=wPaper;
    MoveL Offs(pOrigin,293.04,83.55,6.00),vTravel,z5,tPen\WObj:=wPaper;
    MoveL Offs(pOrigin,293.04,83.55,0.00),v60,z0,tPen\WObj:=wPaper;
    MoveL Offs(pOrigin,287.78,88.81,0.00),v40,z0,tPen\WObj:=wPaper;
    MoveL Offs(pOrigin,288.89,88.92,0.00),v40,z0,tPen\WObj:=wPaper;
    MoveL Offs(pOrigin,289.95,88.92,0.00),v40,z0,tPen\WObj:=wPaper;
    MoveL Offs(pOrigin,290.16,89.98,0.00),v40,z0,tPen\WObj:=wPaper;
    MoveL Offs(pOrigin,289.10,89.98,0.00),v40,z0,tPen\WObj:=wPaper;
    MoveL Offs(pOrigin,289.31,91.03,0.00),v40,z0,tPen\WObj:=wPaper;
    MoveL Offs(pOrigin,290.59,91.03,0.00),v40,z0,tPen\WObj:=wPaper;
    MoveL Offs(pOrigin,290.80,92.09,0.00),v40,z0,tPen\WObj:=wPaper;
    MoveL Offs(pOrigin,289.52,92.09,0.00),v40,z0,tPen\WObj:=wPaper;
    MoveL Offs(pOrigin,289.74,93.14,0.00),v40,z0,tPen\WObj:=wPaper;
    MoveL Offs(pOrigin,291.23,93.14,0.00),v40,fine,tPen\WObj:=wPaper;
    MoveL Offs(pOrigin,291.23,93.14,6.00),v60,z5,tPen\WObj:=wPaper;
    MoveL Offs(pOrigin,291.86,95.26,6.00),vTravel,z5,tPen\WObj:=wPaper;
    MoveL Offs(pOrigin,291.86,95.26,0.00),v60,z0,tPen\WObj:=wPaper;
    MoveL Offs(pOrigin,290.38,95.26,0.00),v40,fine,tPen\WObj:=wPaper;
    MoveL Offs(pOrigin,290.38,95.26,6.00),v60,z5,tPen\WObj:=wPaper;
    MoveL Offs(pOrigin,291.47,97.01,6.00),vTravel,z5,tPen\WObj:=wPaper;
    MoveL Offs(pOrigin,291.47,97.01,0.00),v60,z0,tPen\WObj:=wPaper;
    MoveL Offs(pOrigin,291.47,98.29,0.00),v40,z0,tPen\WObj:=wPaper;
    MoveL Offs(pOrigin,291.23,98.42,0.00),v40,z0,tPen\WObj:=wPaper;
    MoveL Offs(pOrigin,292.71,98.42,0.00),v40,z0,tPen\WObj:=wPaper;
    MoveL Offs(pOrigin,292.50,97.37,0.00),v40,z0,tPen\WObj:=wPaper;
    MoveL Offs(pOrigin,290.80,97.37,0.00),v40,fine,tPen\WObj:=wPaper;
    MoveL Offs(pOrigin,290.80,97.37,6.00),v60,z5,tPen\WObj:=wPaper;
    MoveL Offs(pOrigin,289.99,98.54,6.00),vTravel,z5,tPen\WObj:=wPaper;
    MoveL Offs(pOrigin,289.99,98.54,0.00),v60,z0,tPen\WObj:=wPaper;
    MoveL Offs(pOrigin,293.30,95.24,0.00),v40,fine,tPen\WObj:=wPaper;
    MoveL Offs(pOrigin,293.30,95.24,6.00),v60,z5,tPen\WObj:=wPaper;
    MoveL Offs(pOrigin,293.44,96.58,6.00),vTravel,z5,tPen\WObj:=wPaper;
    MoveL Offs(pOrigin,293.44,96.58,0.00),v60,z0,tPen\WObj:=wPaper;
    MoveL Offs(pOrigin,290.14,99.89,0.00),v40,z0,tPen\WObj:=wPaper;
    MoveL Offs(pOrigin,290.58,99.71,0.00),v40,z0,tPen\WObj:=wPaper;
    MoveL Offs(pOrigin,293.88,103.02,0.00),v40,z0,tPen\WObj:=wPaper;
    MoveL Offs(pOrigin,293.56,102.65,0.00),v40,z0,tPen\WObj:=wPaper;
    MoveL Offs(pOrigin,292.29,102.65,0.00),v40,z0,tPen\WObj:=wPaper;
    MoveL Offs(pOrigin,292.08,101.59,0.00),v40,z0,tPen\WObj:=wPaper;
    MoveL Offs(pOrigin,293.14,101.59,0.00),v40,z0,tPen\WObj:=wPaper;
    MoveL Offs(pOrigin,294.33,101.67,0.00),v40,z0,tPen\WObj:=wPaper;
    MoveL Offs(pOrigin,291.62,104.38,0.00),v40,z0,tPen\WObj:=wPaper;
    MoveL Offs(pOrigin,291.94,104.06,0.00),v40,z0,tPen\WObj:=wPaper;
    MoveL Offs(pOrigin,295.39,107.52,0.00),v40,z0,tPen\WObj:=wPaper;
    MoveL Offs(pOrigin,295.05,107.93,0.00),v40,z0,tPen\WObj:=wPaper;
    MoveL Offs(pOrigin,293.77,107.93,0.00),v40,z0,tPen\WObj:=wPaper;
    MoveL Offs(pOrigin,293.56,106.87,0.00),v40,z0,tPen\WObj:=wPaper;
    MoveL Offs(pOrigin,295.05,106.87,0.00),v40,z0,tPen\WObj:=wPaper;
    MoveL Offs(pOrigin,295.48,105.82,0.00),v40,z0,tPen\WObj:=wPaper;
    MoveL Offs(pOrigin,293.14,105.82,0.00),v40,z0,tPen\WObj:=wPaper;
    MoveL Offs(pOrigin,293.58,105.30,0.00),v40,z0,tPen\WObj:=wPaper;
    MoveL Offs(pOrigin,293.58,106.36,0.00),v40,z0,tPen\WObj:=wPaper;
    MoveL Offs(pOrigin,292.54,106.16,0.00),v40,z0,tPen\WObj:=wPaper;
    MoveL Offs(pOrigin,296.00,109.62,0.00),v40,z0,tPen\WObj:=wPaper;
    MoveL Offs(pOrigin,295.69,110.04,0.00),v40,z0,tPen\WObj:=wPaper;
    MoveL Offs(pOrigin,294.62,110.04,0.00),v40,z0,tPen\WObj:=wPaper;
    MoveL Offs(pOrigin,293.91,110.51,0.00),v40,z0,tPen\WObj:=wPaper;
    MoveL Offs(pOrigin,297.36,113.97,0.00),v40,z0,tPen\WObj:=wPaper;
    MoveL Offs(pOrigin,296.96,114.26,0.00),v40,z0,tPen\WObj:=wPaper;
    MoveL Offs(pOrigin,295.90,114.26,0.00),v40,z0,tPen\WObj:=wPaper;
    MoveL Offs(pOrigin,296.32,115.32,0.00),v40,z0,tPen\WObj:=wPaper;
    MoveL Offs(pOrigin,297.60,115.32,0.00),v40,z0,tPen\WObj:=wPaper;
    MoveL Offs(pOrigin,298.03,114.40,0.00),v40,z0,tPen\WObj:=wPaper;
    MoveL Offs(pOrigin,295.63,116.80,0.00),v40,z0,tPen\WObj:=wPaper;
    MoveL Offs(pOrigin,295.18,115.75,0.00),v40,z0,tPen\WObj:=wPaper;
    MoveL Offs(pOrigin,297.59,113.35,0.00),v40,z0,tPen\WObj:=wPaper;
    MoveL Offs(pOrigin,296.75,113.21,0.00),v40,z0,tPen\WObj:=wPaper;
    MoveL Offs(pOrigin,295.48,113.21,0.00),v40,z0,tPen\WObj:=wPaper;
    MoveL Offs(pOrigin,294.59,113.36,0.00),v40,z0,tPen\WObj:=wPaper;
    MoveL Offs(pOrigin,297.00,110.95,0.00),v40,z0,tPen\WObj:=wPaper;
    MoveL Offs(pOrigin,296.11,111.10,0.00),v40,z0,tPen\WObj:=wPaper;
    MoveL Offs(pOrigin,294.84,111.10,0.00),v40,z0,tPen\WObj:=wPaper;
    MoveL Offs(pOrigin,295.26,112.15,0.00),v40,z0,tPen\WObj:=wPaper;
    MoveL Offs(pOrigin,296.32,112.15,0.00),v40,fine,tPen\WObj:=wPaper;
    MoveL Offs(pOrigin,296.32,112.15,6.00),v60,z5,tPen\WObj:=wPaper;
    MoveL Offs(pOrigin,294.51,112.61,6.00),vTravel,z5,tPen\WObj:=wPaper;
    MoveL Offs(pOrigin,294.51,112.61,0.00),v60,z0,tPen\WObj:=wPaper;
    MoveL Offs(pOrigin,300.07,118.17,0.00),v40,fine,tPen\WObj:=wPaper;
    MoveL Offs(pOrigin,300.07,118.17,6.00),v60,z5,tPen\WObj:=wPaper;
    MoveL Offs(pOrigin,298.88,117.43,6.00),vTravel,z5,tPen\WObj:=wPaper;
  ENDPROC

  PROC DrawPart134()
    MoveL Offs(pOrigin,298.88,117.43,0.00),v60,z0,tPen\WObj:=wPaper;
    MoveL Offs(pOrigin,296.75,117.43,0.00),v40,z0,tPen\WObj:=wPaper;
    MoveL Offs(pOrigin,295.93,118.00,0.00),v40,z0,tPen\WObj:=wPaper;
    MoveL Offs(pOrigin,298.78,115.14,0.00),v40,fine,tPen\WObj:=wPaper;
    MoveL Offs(pOrigin,298.78,115.14,6.00),v60,z5,tPen\WObj:=wPaper;
    MoveL Offs(pOrigin,301.93,114.98,6.00),vTravel,z5,tPen\WObj:=wPaper;
    MoveL Offs(pOrigin,301.93,114.98,0.00),v60,z0,tPen\WObj:=wPaper;
    MoveL Offs(pOrigin,296.67,120.24,0.00),v40,fine,tPen\WObj:=wPaper;
    MoveL Offs(pOrigin,296.67,120.24,6.00),v60,z5,tPen\WObj:=wPaper;
    MoveL Offs(pOrigin,300.56,122.33,6.00),vTravel,z5,tPen\WObj:=wPaper;
    MoveL Offs(pOrigin,300.56,122.33,0.00),v60,z0,tPen\WObj:=wPaper;
    MoveL Offs(pOrigin,298.15,124.73,0.00),v40,fine,tPen\WObj:=wPaper;
    MoveL Offs(pOrigin,298.15,124.73,6.00),v60,z5,tPen\WObj:=wPaper;
    MoveL Offs(pOrigin,299.51,125.88,6.00),vTravel,z5,tPen\WObj:=wPaper;
    MoveL Offs(pOrigin,299.51,125.88,0.00),v60,z0,tPen\WObj:=wPaper;
    MoveL Offs(pOrigin,300.58,125.88,0.00),v40,z0,tPen\WObj:=wPaper;
    MoveL Offs(pOrigin,301.59,125.77,0.00),v40,z0,tPen\WObj:=wPaper;
    MoveL Offs(pOrigin,299.19,128.17,0.00),v40,z0,tPen\WObj:=wPaper;
    MoveL Offs(pOrigin,299.35,127.90,0.00),v40,z0,tPen\WObj:=wPaper;
    MoveL Offs(pOrigin,302.81,131.36,0.00),v40,z0,tPen\WObj:=wPaper;
    MoveL Offs(pOrigin,302.27,131.16,0.00),v40,z0,tPen\WObj:=wPaper;
    MoveL Offs(pOrigin,301.21,131.16,0.00),v40,z0,tPen\WObj:=wPaper;
    MoveL Offs(pOrigin,300.23,131.62,0.00),v40,z0,tPen\WObj:=wPaper;
    MoveL Offs(pOrigin,302.63,129.21,0.00),v40,fine,tPen\WObj:=wPaper;
    MoveL Offs(pOrigin,302.63,129.21,6.00),v60,z5,tPen\WObj:=wPaper;
    MoveL Offs(pOrigin,303.37,131.46,6.00),vTravel,z5,tPen\WObj:=wPaper;
    MoveL Offs(pOrigin,303.37,131.46,0.00),v60,z0,tPen\WObj:=wPaper;
    MoveL Offs(pOrigin,300.82,134.01,0.00),v40,fine,tPen\WObj:=wPaper;
    MoveL Offs(pOrigin,300.82,134.01,6.00),v60,z5,tPen\WObj:=wPaper;
    MoveL Offs(pOrigin,301.86,137.45,6.00),vTravel,z5,tPen\WObj:=wPaper;
    MoveL Offs(pOrigin,301.86,137.45,0.00),v60,z0,tPen\WObj:=wPaper;
    MoveL Offs(pOrigin,304.41,134.90,0.00),v40,fine,tPen\WObj:=wPaper;
    MoveL Offs(pOrigin,304.41,134.90,6.00),v60,z5,tPen\WObj:=wPaper;
    MoveL Offs(pOrigin,304.71,136.10,6.00),vTravel,z5,tPen\WObj:=wPaper;
    MoveL Offs(pOrigin,304.71,136.10,0.00),v60,z0,tPen\WObj:=wPaper;
    MoveL Offs(pOrigin,302.30,138.50,0.00),v40,z0,tPen\WObj:=wPaper;
    MoveL Offs(pOrigin,302.98,139.00,0.00),v40,z0,tPen\WObj:=wPaper;
    MoveL Offs(pOrigin,306.29,142.30,0.00),v40,z0,tPen\WObj:=wPaper;
    MoveL Offs(pOrigin,306.49,141.78,0.00),v40,z0,tPen\WObj:=wPaper;
    MoveL Offs(pOrigin,304.08,144.19,0.00),v40,z0,tPen\WObj:=wPaper;
    MoveL Offs(pOrigin,304.53,145.23,0.00),v40,z0,tPen\WObj:=wPaper;
    MoveL Offs(pOrigin,306.93,142.83,0.00),v40,z0,tPen\WObj:=wPaper;
    MoveL Offs(pOrigin,305.89,142.78,0.00),v40,z0,tPen\WObj:=wPaper;
    MoveL Offs(pOrigin,304.82,142.78,0.00),v40,fine,tPen\WObj:=wPaper;
    MoveL Offs(pOrigin,304.82,142.78,6.00),v60,z5,tPen\WObj:=wPaper;
    MoveL Offs(pOrigin,307.38,143.88,6.00),vTravel,z5,tPen\WObj:=wPaper;
    MoveL Offs(pOrigin,307.38,143.88,0.00),v60,z0,tPen\WObj:=wPaper;
    MoveL Offs(pOrigin,304.83,146.43,0.00),v40,z0,tPen\WObj:=wPaper;
    MoveL Offs(pOrigin,305.89,145.94,0.00),v40,z0,tPen\WObj:=wPaper;
    MoveL Offs(pOrigin,306.95,145.94,0.00),v40,z0,tPen\WObj:=wPaper;
    MoveL Offs(pOrigin,307.53,145.23,0.00),v40,z0,tPen\WObj:=wPaper;
    MoveL Offs(pOrigin,305.12,147.63,0.00),v40,fine,tPen\WObj:=wPaper;
    MoveL Offs(pOrigin,305.12,147.63,6.00),v60,z5,tPen\WObj:=wPaper;
    MoveL Offs(pOrigin,311.42,145.81,6.00),vTravel,z5,tPen\WObj:=wPaper;
    MoveL Offs(pOrigin,311.42,145.81,0.00),v60,z0,tPen\WObj:=wPaper;
    MoveL Offs(pOrigin,312.32,144.91,0.00),v40,z0,tPen\WObj:=wPaper;
    MoveL Offs(pOrigin,312.92,145.81,0.00),v40,z0,tPen\WObj:=wPaper;
    MoveL Offs(pOrigin,311.72,147.01,0.00),v40,z0,tPen\WObj:=wPaper;
    MoveL Offs(pOrigin,312.46,147.76,0.00),v40,z0,tPen\WObj:=wPaper;
    MoveL Offs(pOrigin,313.36,146.86,0.00),v40,z0,tPen\WObj:=wPaper;
    MoveL Offs(pOrigin,313.96,147.75,0.00),v40,z0,tPen\WObj:=wPaper;
    MoveL Offs(pOrigin,312.76,148.95,0.00),v40,z0,tPen\WObj:=wPaper;
    MoveL Offs(pOrigin,313.35,149.85,0.00),v40,z0,tPen\WObj:=wPaper;
    MoveL Offs(pOrigin,314.56,148.65,0.00),v40,z0,tPen\WObj:=wPaper;
    MoveL Offs(pOrigin,315.00,149.70,0.00),v40,z0,tPen\WObj:=wPaper;
    MoveL Offs(pOrigin,313.80,150.90,0.00),v40,z0,tPen\WObj:=wPaper;
    MoveL Offs(pOrigin,314.40,151.80,0.00),v40,z0,tPen\WObj:=wPaper;
    MoveL Offs(pOrigin,315.60,150.59,0.00),v40,z0,tPen\WObj:=wPaper;
    MoveL Offs(pOrigin,316.20,151.49,0.00),v40,z0,tPen\WObj:=wPaper;
    MoveL Offs(pOrigin,314.99,152.69,0.00),v40,z0,tPen\WObj:=wPaper;
    MoveL Offs(pOrigin,315.44,153.74,0.00),v40,z0,tPen\WObj:=wPaper;
    MoveL Offs(pOrigin,316.79,152.39,0.00),v40,z0,tPen\WObj:=wPaper;
    MoveL Offs(pOrigin,317.39,153.28,0.00),v40,z0,tPen\WObj:=wPaper;
    MoveL Offs(pOrigin,316.04,154.64,0.00),v40,z0,tPen\WObj:=wPaper;
    MoveL Offs(pOrigin,316.63,155.53,0.00),v40,z0,tPen\WObj:=wPaper;
    MoveL Offs(pOrigin,317.99,154.18,0.00),v40,z0,tPen\WObj:=wPaper;
    MoveL Offs(pOrigin,317.15,154.39,0.00),v40,z0,tPen\WObj:=wPaper;
    MoveL Offs(pOrigin,317.36,154.81,0.00),v40,z0,tPen\WObj:=wPaper;
    MoveL Offs(pOrigin,317.15,154.39,0.00),v40,z0,tPen\WObj:=wPaper;
    MoveL Offs(pOrigin,316.73,153.75,0.00),v40,z0,tPen\WObj:=wPaper;
    MoveL Offs(pOrigin,316.94,154.18,0.00),v40,z0,tPen\WObj:=wPaper;
    MoveL Offs(pOrigin,316.73,153.75,0.00),v40,fine,tPen\WObj:=wPaper;
    MoveL Offs(pOrigin,316.73,153.75,6.00),v60,z5,tPen\WObj:=wPaper;
    MoveL Offs(pOrigin,318.58,155.08,6.00),vTravel,z5,tPen\WObj:=wPaper;
    MoveL Offs(pOrigin,318.58,155.08,0.00),v60,z0,tPen\WObj:=wPaper;
    MoveL Offs(pOrigin,317.23,156.43,0.00),v40,z0,tPen\WObj:=wPaper;
    MoveL Offs(pOrigin,317.68,157.48,0.00),v40,z0,tPen\WObj:=wPaper;
    MoveL Offs(pOrigin,319.18,155.98,0.00),v40,z0,tPen\WObj:=wPaper;
    MoveL Offs(pOrigin,319.77,156.87,0.00),v40,z0,tPen\WObj:=wPaper;
    MoveL Offs(pOrigin,318.27,158.37,0.00),v40,z0,tPen\WObj:=wPaper;
    MoveL Offs(pOrigin,318.92,157.92,0.00),v40,z0,tPen\WObj:=wPaper;
    MoveL Offs(pOrigin,321.62,160.63,0.00),v40,z0,tPen\WObj:=wPaper;
    MoveL Offs(pOrigin,322.16,160.46,0.00),v40,z0,tPen\WObj:=wPaper;
    MoveL Offs(pOrigin,320.81,161.81,0.00),v40,z0,tPen\WObj:=wPaper;
    MoveL Offs(pOrigin,321.48,161.97,0.00),v40,z0,tPen\WObj:=wPaper;
    MoveL Offs(pOrigin,327.19,167.68,0.00),v40,z0,tPen\WObj:=wPaper;
    MoveL Offs(pOrigin,327.53,167.03,0.00),v40,z0,tPen\WObj:=wPaper;
    MoveL Offs(pOrigin,326.03,168.54,0.00),v40,z0,tPen\WObj:=wPaper;
    MoveL Offs(pOrigin,325.28,167.79,0.00),v40,z0,tPen\WObj:=wPaper;
    MoveL Offs(pOrigin,326.79,166.29,0.00),v40,z0,tPen\WObj:=wPaper;
    MoveL Offs(pOrigin,326.19,165.39,0.00),v40,z0,tPen\WObj:=wPaper;
    MoveL Offs(pOrigin,324.69,166.89,0.00),v40,z0,tPen\WObj:=wPaper;
    MoveL Offs(pOrigin,323.94,166.15,0.00),v40,z0,tPen\WObj:=wPaper;
    MoveL Offs(pOrigin,325.59,164.49,0.00),v40,z0,tPen\WObj:=wPaper;
    MoveL Offs(pOrigin,324.85,163.75,0.00),v40,z0,tPen\WObj:=wPaper;
    MoveL Offs(pOrigin,323.19,165.40,0.00),v40,z0,tPen\WObj:=wPaper;
    MoveL Offs(pOrigin,322.60,164.50,0.00),v40,z0,tPen\WObj:=wPaper;
    MoveL Offs(pOrigin,324.10,163.00,0.00),v40,z0,tPen\WObj:=wPaper;
    MoveL Offs(pOrigin,323.50,162.10,0.00),v40,z0,tPen\WObj:=wPaper;
    MoveL Offs(pOrigin,322.00,163.61,0.00),v40,z0,tPen\WObj:=wPaper;
    MoveL Offs(pOrigin,321.25,162.86,0.00),v40,z0,tPen\WObj:=wPaper;
    MoveL Offs(pOrigin,322.91,161.21,0.00),v40,fine,tPen\WObj:=wPaper;
    MoveL Offs(pOrigin,322.91,161.21,6.00),v60,z5,tPen\WObj:=wPaper;
    MoveL Offs(pOrigin,321.56,159.56,6.00),vTravel,z5,tPen\WObj:=wPaper;
    MoveL Offs(pOrigin,321.56,159.56,0.00),v60,z0,tPen\WObj:=wPaper;
    MoveL Offs(pOrigin,320.21,160.92,0.00),v40,z0,tPen\WObj:=wPaper;
    MoveL Offs(pOrigin,319.62,160.02,0.00),v40,z0,tPen\WObj:=wPaper;
    MoveL Offs(pOrigin,321.12,158.52,0.00),v40,z0,tPen\WObj:=wPaper;
    MoveL Offs(pOrigin,320.52,157.62,0.00),v40,z0,tPen\WObj:=wPaper;
    MoveL Offs(pOrigin,318.87,159.27,0.00),v40,fine,tPen\WObj:=wPaper;
  ENDPROC

  PROC DrawPart135()
    MoveL Offs(pOrigin,318.87,159.27,6.00),v60,z5,tPen\WObj:=wPaper;
    MoveL Offs(pOrigin,313.31,163.33,6.00),vTravel,z5,tPen\WObj:=wPaper;
    MoveL Offs(pOrigin,313.31,163.33,0.00),v60,z0,tPen\WObj:=wPaper;
    MoveL Offs(pOrigin,310.91,165.74,0.00),v40,z0,tPen\WObj:=wPaper;
    MoveL Offs(pOrigin,311.36,166.78,0.00),v40,z0,tPen\WObj:=wPaper;
    MoveL Offs(pOrigin,313.61,164.53,0.00),v40,z0,tPen\WObj:=wPaper;
    MoveL Offs(pOrigin,313.09,164.05,0.00),v40,z0,tPen\WObj:=wPaper;
    MoveL Offs(pOrigin,309.94,160.89,0.00),v40,z0,tPen\WObj:=wPaper;
    MoveL Offs(pOrigin,309.42,161.25,0.00),v40,z0,tPen\WObj:=wPaper;
    MoveL Offs(pOrigin,311.98,158.69,0.00),v40,z0,tPen\WObj:=wPaper;
    MoveL Offs(pOrigin,311.53,157.65,0.00),v40,z0,tPen\WObj:=wPaper;
    MoveL Offs(pOrigin,309.13,160.05,0.00),v40,z0,tPen\WObj:=wPaper;
    MoveL Offs(pOrigin,310.14,159.67,0.00),v40,z0,tPen\WObj:=wPaper;
    MoveL Offs(pOrigin,311.20,159.67,0.00),v40,fine,tPen\WObj:=wPaper;
    MoveL Offs(pOrigin,311.20,159.67,6.00),v60,z5,tPen\WObj:=wPaper;
    MoveL Offs(pOrigin,310.14,156.50,6.00),vTravel,z5,tPen\WObj:=wPaper;
    MoveL Offs(pOrigin,310.14,156.50,0.00),v60,z0,tPen\WObj:=wPaper;
    MoveL Offs(pOrigin,309.08,156.50,0.00),v40,fine,tPen\WObj:=wPaper;
    MoveL Offs(pOrigin,309.08,156.50,6.00),v60,z5,tPen\WObj:=wPaper;
    MoveL Offs(pOrigin,311.84,164.95,6.00),vTravel,z5,tPen\WObj:=wPaper;
    MoveL Offs(pOrigin,311.84,164.95,0.00),v60,z0,tPen\WObj:=wPaper;
    MoveL Offs(pOrigin,312.90,164.95,0.00),v40,fine,tPen\WObj:=wPaper;
    MoveL Offs(pOrigin,312.90,164.95,6.00),v60,z5,tPen\WObj:=wPaper;
    MoveL Offs(pOrigin,314.50,166.63,6.00),vTravel,z5,tPen\WObj:=wPaper;
    MoveL Offs(pOrigin,314.50,166.63,0.00),v60,z0,tPen\WObj:=wPaper;
    MoveL Offs(pOrigin,311.95,169.18,0.00),v40,fine,tPen\WObj:=wPaper;
    MoveL Offs(pOrigin,311.95,169.18,6.00),v60,z5,tPen\WObj:=wPaper;
    MoveL Offs(pOrigin,315.99,171.11,6.00),vTravel,z5,tPen\WObj:=wPaper;
    MoveL Offs(pOrigin,315.99,171.11,0.00),v60,z0,tPen\WObj:=wPaper;
    MoveL Offs(pOrigin,313.58,173.52,0.00),v40,fine,tPen\WObj:=wPaper;
    MoveL Offs(pOrigin,313.58,173.52,6.00),v60,z5,tPen\WObj:=wPaper;
    MoveL Offs(pOrigin,315.02,174.46,6.00),vTravel,z5,tPen\WObj:=wPaper;
    MoveL Offs(pOrigin,315.02,174.46,0.00),v60,z0,tPen\WObj:=wPaper;
    MoveL Offs(pOrigin,316.09,174.46,0.00),v40,z0,tPen\WObj:=wPaper;
    MoveL Offs(pOrigin,316.58,173.51,0.00),v40,z0,tPen\WObj:=wPaper;
    MoveL Offs(pOrigin,314.17,175.91,0.00),v40,fine,tPen\WObj:=wPaper;
    MoveL Offs(pOrigin,314.17,175.91,6.00),v60,z5,tPen\WObj:=wPaper;
    MoveL Offs(pOrigin,317.15,180.79,6.00),vTravel,z5,tPen\WObj:=wPaper;
    MoveL Offs(pOrigin,317.15,180.79,0.00),v60,z0,tPen\WObj:=wPaper;
    MoveL Offs(pOrigin,318.21,180.79,0.00),v40,fine,tPen\WObj:=wPaper;
    MoveL Offs(pOrigin,318.21,180.79,6.00),v60,z5,tPen\WObj:=wPaper;
    MoveL Offs(pOrigin,320.55,182.01,6.00),vTravel,z5,tPen\WObj:=wPaper;
    MoveL Offs(pOrigin,320.55,182.01,0.00),v60,z0,tPen\WObj:=wPaper;
    MoveL Offs(pOrigin,320.34,183.29,0.00),v40,z0,tPen\WObj:=wPaper;
    MoveL Offs(pOrigin,320.55,183.50,0.00),v40,z0,tPen\WObj:=wPaper;
    MoveL Offs(pOrigin,320.55,183.50,0.00),v40,z0,tPen\WObj:=wPaper;
    MoveL Offs(pOrigin,320.55,184.56,0.00),v40,z0,tPen\WObj:=wPaper;
    MoveL Offs(pOrigin,320.55,184.56,0.00),v40,z0,tPen\WObj:=wPaper;
    MoveL Offs(pOrigin,320.98,185.20,0.00),v40,z0,tPen\WObj:=wPaper;
    MoveL Offs(pOrigin,320.41,186.05,0.00),v40,z0,tPen\WObj:=wPaper;
    MoveL Offs(pOrigin,318.71,191.57,0.00),v40,z0,tPen\WObj:=wPaper;
    MoveL Offs(pOrigin,316.80,194.55,0.00),v40,z0,tPen\WObj:=wPaper;
    MoveL Offs(pOrigin,313.18,198.59,0.00),v40,z0,tPen\WObj:=wPaper;
    MoveL Offs(pOrigin,309.36,203.90,0.00),v40,z0,tPen\WObj:=wPaper;
    MoveL Offs(pOrigin,309.92,204.11,0.00),v40,z0,tPen\WObj:=wPaper;
    MoveL Offs(pOrigin,313.96,203.26,0.00),v40,z0,tPen\WObj:=wPaper;
    MoveL Offs(pOrigin,321.61,201.14,0.00),v40,z0,tPen\WObj:=wPaper;
    MoveL Offs(pOrigin,322.25,201.35,0.00),v40,z0,tPen\WObj:=wPaper;
    MoveL Offs(pOrigin,322.25,201.35,0.00),v40,z0,tPen\WObj:=wPaper;
    MoveL Offs(pOrigin,336.27,196.46,0.00),v40,z0,tPen\WObj:=wPaper;
    MoveL Offs(pOrigin,337.34,196.46,0.00),v40,fine,tPen\WObj:=wPaper;
    MoveL Offs(pOrigin,337.34,196.46,6.00),v60,z5,tPen\WObj:=wPaper;
    MoveL Offs(pOrigin,329.84,197.59,6.00),vTravel,z5,tPen\WObj:=wPaper;
    MoveL Offs(pOrigin,329.84,197.59,0.00),v60,z0,tPen\WObj:=wPaper;
    MoveL Offs(pOrigin,326.53,200.89,0.00),v40,fine,tPen\WObj:=wPaper;
    MoveL Offs(pOrigin,326.53,200.89,6.00),v60,z5,tPen\WObj:=wPaper;
    MoveL Offs(pOrigin,325.34,199.10,6.00),vTravel,z5,tPen\WObj:=wPaper;
    MoveL Offs(pOrigin,325.34,199.10,0.00),v60,z0,tPen\WObj:=wPaper;
    MoveL Offs(pOrigin,321.88,202.55,0.00),v40,z0,tPen\WObj:=wPaper;
    MoveL Offs(pOrigin,321.30,202.12,0.00),v40,z0,tPen\WObj:=wPaper;
    MoveL Offs(pOrigin,320.55,201.37,0.00),v40,z0,tPen\WObj:=wPaper;
    MoveL Offs(pOrigin,319.50,201.82,0.00),v40,z0,tPen\WObj:=wPaper;
    MoveL Offs(pOrigin,320.25,202.57,0.00),v40,z0,tPen\WObj:=wPaper;
    MoveL Offs(pOrigin,319.48,203.46,0.00),v40,z0,tPen\WObj:=wPaper;
    MoveL Offs(pOrigin,323.24,199.70,0.00),v40,fine,tPen\WObj:=wPaper;
    MoveL Offs(pOrigin,323.24,199.70,6.00),v60,z5,tPen\WObj:=wPaper;
    MoveL Offs(pOrigin,321.14,200.31,6.00),vTravel,z5,tPen\WObj:=wPaper;
    MoveL Offs(pOrigin,321.14,200.31,0.00),v60,z0,tPen\WObj:=wPaper;
    MoveL Offs(pOrigin,317.38,204.07,0.00),v40,z0,tPen\WObj:=wPaper;
    MoveL Offs(pOrigin,316.96,203.75,0.00),v40,z0,tPen\WObj:=wPaper;
    MoveL Offs(pOrigin,315.91,202.70,0.00),v40,fine,tPen\WObj:=wPaper;
    MoveL Offs(pOrigin,315.91,202.70,6.00),v60,z5,tPen\WObj:=wPaper;
    MoveL Offs(pOrigin,314.84,202.13,6.00),vTravel,z5,tPen\WObj:=wPaper;
    MoveL Offs(pOrigin,314.84,202.13,0.00),v60,z0,tPen\WObj:=wPaper;
    MoveL Offs(pOrigin,311.69,205.28,0.00),v40,z0,tPen\WObj:=wPaper;
    MoveL Offs(pOrigin,312.02,204.79,0.00),v40,z0,tPen\WObj:=wPaper;
    MoveL Offs(pOrigin,308.87,201.63,0.00),v40,z0,tPen\WObj:=wPaper;
    MoveL Offs(pOrigin,309.08,201.91,0.00),v40,z0,tPen\WObj:=wPaper;
    MoveL Offs(pOrigin,310.35,201.91,0.00),v40,z0,tPen\WObj:=wPaper;
    MoveL Offs(pOrigin,310.35,201.99,0.00),v40,z0,tPen\WObj:=wPaper;
    MoveL Offs(pOrigin,309.92,202.62,0.00),v40,z0,tPen\WObj:=wPaper;
    MoveL Offs(pOrigin,310.35,201.99,0.00),v40,z0,tPen\WObj:=wPaper;
    MoveL Offs(pOrigin,310.81,202.09,0.00),v40,z0,tPen\WObj:=wPaper;
    MoveL Offs(pOrigin,309.46,200.74,0.00),v40,z0,tPen\WObj:=wPaper;
    MoveL Offs(pOrigin,309.92,200.86,0.00),v40,z0,tPen\WObj:=wPaper;
    MoveL Offs(pOrigin,311.20,200.86,0.00),v40,z0,tPen\WObj:=wPaper;
    MoveL Offs(pOrigin,311.41,201.19,0.00),v40,z0,tPen\WObj:=wPaper;
    MoveL Offs(pOrigin,310.06,199.84,0.00),v40,z0,tPen\WObj:=wPaper;
    MoveL Offs(pOrigin,310.14,200.07,0.00),v40,z0,tPen\WObj:=wPaper;
    MoveL Offs(pOrigin,309.71,200.50,0.00),v40,z0,tPen\WObj:=wPaper;
    MoveL Offs(pOrigin,310.14,200.07,0.00),v40,z0,tPen\WObj:=wPaper;
    MoveL Offs(pOrigin,310.56,199.80,0.00),v40,z0,tPen\WObj:=wPaper;
    MoveL Offs(pOrigin,312.05,199.80,0.00),v40,z0,tPen\WObj:=wPaper;
    MoveL Offs(pOrigin,312.01,200.29,0.00),v40,z0,tPen\WObj:=wPaper;
    MoveL Offs(pOrigin,310.65,198.94,0.00),v40,z0,tPen\WObj:=wPaper;
    MoveL Offs(pOrigin,311.20,198.59,0.00),v40,z0,tPen\WObj:=wPaper;
    MoveL Offs(pOrigin,310.77,199.23,0.00),v40,z0,tPen\WObj:=wPaper;
    MoveL Offs(pOrigin,311.20,198.59,0.00),v40,z0,tPen\WObj:=wPaper;
    MoveL Offs(pOrigin,311.41,198.74,0.00),v40,z0,tPen\WObj:=wPaper;
    MoveL Offs(pOrigin,312.69,198.74,0.00),v40,z0,tPen\WObj:=wPaper;
    MoveL Offs(pOrigin,313.11,198.38,0.00),v40,z0,tPen\WObj:=wPaper;
    MoveL Offs(pOrigin,312.69,199.01,0.00),v40,z0,tPen\WObj:=wPaper;
    MoveL Offs(pOrigin,313.11,198.38,0.00),v40,z0,tPen\WObj:=wPaper;
    MoveL Offs(pOrigin,313.50,198.80,0.00),v40,z0,tPen\WObj:=wPaper;
    MoveL Offs(pOrigin,312.00,197.30,0.00),v40,z0,tPen\WObj:=wPaper;
    MoveL Offs(pOrigin,312.26,197.69,0.00),v40,z0,tPen\WObj:=wPaper;
    MoveL Offs(pOrigin,313.75,197.69,0.00),v40,z0,tPen\WObj:=wPaper;
    MoveL Offs(pOrigin,314.10,197.90,0.00),v40,z0,tPen\WObj:=wPaper;
    MoveL Offs(pOrigin,312.59,196.40,0.00),v40,z0,tPen\WObj:=wPaper;
    MoveL Offs(pOrigin,312.69,196.89,0.00),v40,z0,tPen\WObj:=wPaper;
  ENDPROC

  PROC DrawPart136()
    MoveL Offs(pOrigin,312.05,197.52,0.00),v40,z0,tPen\WObj:=wPaper;
    MoveL Offs(pOrigin,312.69,196.89,0.00),v40,fine,tPen\WObj:=wPaper;
    MoveL Offs(pOrigin,312.69,196.89,6.00),v60,z5,tPen\WObj:=wPaper;
    MoveL Offs(pOrigin,312.47,195.54,6.00),vTravel,z5,tPen\WObj:=wPaper;
    MoveL Offs(pOrigin,312.47,195.54,0.00),v60,z0,tPen\WObj:=wPaper;
    MoveL Offs(pOrigin,315.02,192.99,0.00),v40,z0,tPen\WObj:=wPaper;
    MoveL Offs(pOrigin,314.60,193.91,0.00),v40,z0,tPen\WObj:=wPaper;
    MoveL Offs(pOrigin,315.02,194.12,0.00),v40,z0,tPen\WObj:=wPaper;
    MoveL Offs(pOrigin,314.60,193.91,0.00),v40,z0,tPen\WObj:=wPaper;
    MoveL Offs(pOrigin,315.45,194.52,0.00),v40,z0,tPen\WObj:=wPaper;
    MoveL Offs(pOrigin,313.32,194.52,0.00),v40,z0,tPen\WObj:=wPaper;
    MoveL Offs(pOrigin,312.69,194.34,0.00),v40,z0,tPen\WObj:=wPaper;
    MoveL Offs(pOrigin,313.11,194.55,0.00),v40,z0,tPen\WObj:=wPaper;
    MoveL Offs(pOrigin,312.69,194.34,0.00),v40,z0,tPen\WObj:=wPaper;
    MoveL Offs(pOrigin,311.72,194.80,0.00),v40,z0,tPen\WObj:=wPaper;
    MoveL Offs(pOrigin,313.97,192.54,0.00),v40,fine,tPen\WObj:=wPaper;
    MoveL Offs(pOrigin,313.97,192.54,6.00),v60,z5,tPen\WObj:=wPaper;
    MoveL Offs(pOrigin,311.20,192.41,6.00),vTravel,z5,tPen\WObj:=wPaper;
    MoveL Offs(pOrigin,311.20,192.41,0.00),v60,z0,tPen\WObj:=wPaper;
    MoveL Offs(pOrigin,309.08,192.41,0.00),v40,z0,tPen\WObj:=wPaper;
    MoveL Offs(pOrigin,308.73,193.31,0.00),v40,z0,tPen\WObj:=wPaper;
    MoveL Offs(pOrigin,310.98,191.05,0.00),v40,z0,tPen\WObj:=wPaper;
    MoveL Offs(pOrigin,310.78,191.60,0.00),v40,z0,tPen\WObj:=wPaper;
    MoveL Offs(pOrigin,315.59,196.41,0.00),v40,fine,tPen\WObj:=wPaper;
    MoveL Offs(pOrigin,315.59,196.41,6.00),v60,z5,tPen\WObj:=wPaper;
    MoveL Offs(pOrigin,316.09,194.98,6.00),vTravel,z5,tPen\WObj:=wPaper;
    MoveL Offs(pOrigin,316.09,194.98,0.00),v60,z0,tPen\WObj:=wPaper;
    MoveL Offs(pOrigin,314.39,193.56,0.00),v40,z0,tPen\WObj:=wPaper;
    MoveL Offs(pOrigin,306.95,190.16,0.00),v40,z0,tPen\WObj:=wPaper;
    MoveL Offs(pOrigin,303.90,188.39,0.00),v40,z0,tPen\WObj:=wPaper;
    MoveL Offs(pOrigin,304.40,187.89,0.00),v40,z0,tPen\WObj:=wPaper;
    MoveL Offs(pOrigin,318.21,183.15,0.00),v40,z0,tPen\WObj:=wPaper;
    MoveL Offs(pOrigin,318.64,182.65,0.00),v40,z0,tPen\WObj:=wPaper;
    MoveL Offs(pOrigin,318.64,181.59,0.00),v40,z0,tPen\WObj:=wPaper;
    MoveL Offs(pOrigin,310.35,156.51,0.00),v40,z0,tPen\WObj:=wPaper;
    MoveL Offs(pOrigin,298.38,117.62,0.00),v40,z0,tPen\WObj:=wPaper;
    MoveL Offs(pOrigin,298.66,117.41,0.00),v40,z0,tPen\WObj:=wPaper;
    MoveL Offs(pOrigin,322.04,123.79,0.00),v40,z0,tPen\WObj:=wPaper;
    MoveL Offs(pOrigin,331.60,126.55,0.00),v40,z0,tPen\WObj:=wPaper;
    MoveL Offs(pOrigin,335.00,128.04,0.00),v40,fine,tPen\WObj:=wPaper;
    MoveL Offs(pOrigin,335.00,128.04,6.00),v60,z5,tPen\WObj:=wPaper;
    MoveL Offs(pOrigin,335.85,126.94,6.00),vTravel,z5,tPen\WObj:=wPaper;
    MoveL Offs(pOrigin,335.85,126.94,0.00),v60,z0,tPen\WObj:=wPaper;
    MoveL Offs(pOrigin,333.09,126.94,0.00),v40,z0,tPen\WObj:=wPaper;
    MoveL Offs(pOrigin,332.45,127.77,0.00),v40,z0,tPen\WObj:=wPaper;
    MoveL Offs(pOrigin,336.65,123.57,0.00),v40,z0,tPen\WObj:=wPaper;
    MoveL Offs(pOrigin,336.04,124.27,0.00),v40,z0,tPen\WObj:=wPaper;
    MoveL Offs(pOrigin,336.94,125.17,0.00),v40,fine,tPen\WObj:=wPaper;
    MoveL Offs(pOrigin,336.94,125.17,6.00),v60,z5,tPen\WObj:=wPaper;
    MoveL Offs(pOrigin,336.80,126.52,6.00),vTravel,z5,tPen\WObj:=wPaper;
    MoveL Offs(pOrigin,336.80,126.52,0.00),v60,z0,tPen\WObj:=wPaper;
    MoveL Offs(pOrigin,339.50,129.22,0.00),v40,fine,tPen\WObj:=wPaper;
    MoveL Offs(pOrigin,339.50,129.22,6.00),v60,z5,tPen\WObj:=wPaper;
    MoveL Offs(pOrigin,340.68,129.99,6.00),vTravel,z5,tPen\WObj:=wPaper;
    MoveL Offs(pOrigin,340.68,129.99,0.00),v60,z0,tPen\WObj:=wPaper;
    MoveL Offs(pOrigin,346.39,124.28,0.00),v40,z0,tPen\WObj:=wPaper;
    MoveL Offs(pOrigin,345.93,123.70,0.00),v40,z0,tPen\WObj:=wPaper;
    MoveL Offs(pOrigin,344.42,122.20,0.00),v40,z0,tPen\WObj:=wPaper;
    MoveL Offs(pOrigin,343.85,122.34,0.00),v40,z0,tPen\WObj:=wPaper;
    MoveL Offs(pOrigin,346.40,119.79,0.00),v40,z0,tPen\WObj:=wPaper;
    MoveL Offs(pOrigin,345.92,120.71,0.00),v40,z0,tPen\WObj:=wPaper;
    MoveL Offs(pOrigin,342.46,117.25,0.00),v40,z0,tPen\WObj:=wPaper;
    MoveL Offs(pOrigin,342.22,116.51,0.00),v40,z0,tPen\WObj:=wPaper;
    MoveL Offs(pOrigin,340.27,118.46,0.00),v40,z0,tPen\WObj:=wPaper;
    MoveL Offs(pOrigin,340.22,117.99,0.00),v40,z0,tPen\WObj:=wPaper;
    MoveL Offs(pOrigin,337.96,115.74,0.00),v40,z0,tPen\WObj:=wPaper;
    MoveL Offs(pOrigin,337.73,115.02,0.00),v40,z0,tPen\WObj:=wPaper;
    MoveL Offs(pOrigin,335.78,116.98,0.00),v40,z0,tPen\WObj:=wPaper;
    MoveL Offs(pOrigin,335.87,116.63,0.00),v40,z0,tPen\WObj:=wPaper;
    MoveL Offs(pOrigin,333.76,114.53,0.00),v40,z0,tPen\WObj:=wPaper;
    MoveL Offs(pOrigin,334.29,113.99,0.00),v40,z0,tPen\WObj:=wPaper;
    MoveL Offs(pOrigin,332.33,115.94,0.00),v40,z0,tPen\WObj:=wPaper;
    MoveL Offs(pOrigin,331.67,115.42,0.00),v40,z0,tPen\WObj:=wPaper;
    MoveL Offs(pOrigin,329.42,113.16,0.00),v40,z0,tPen\WObj:=wPaper;
    MoveL Offs(pOrigin,329.80,112.50,0.00),v40,z0,tPen\WObj:=wPaper;
    MoveL Offs(pOrigin,327.69,114.60,0.00),v40,z0,tPen\WObj:=wPaper;
    MoveL Offs(pOrigin,327.62,114.36,0.00),v40,z0,tPen\WObj:=wPaper;
    MoveL Offs(pOrigin,325.37,112.10,0.00),v40,z0,tPen\WObj:=wPaper;
    MoveL Offs(pOrigin,326.05,111.76,0.00),v40,z0,tPen\WObj:=wPaper;
    MoveL Offs(pOrigin,324.10,113.72,0.00),v40,z0,tPen\WObj:=wPaper;
    MoveL Offs(pOrigin,323.27,113.00,0.00),v40,z0,tPen\WObj:=wPaper;
    MoveL Offs(pOrigin,321.32,111.04,0.00),v40,z0,tPen\WObj:=wPaper;
    MoveL Offs(pOrigin,321.41,110.43,0.00),v40,z0,tPen\WObj:=wPaper;
    MoveL Offs(pOrigin,319.46,112.38,0.00),v40,z0,tPen\WObj:=wPaper;
    MoveL Offs(pOrigin,319.23,111.93,0.00),v40,z0,tPen\WObj:=wPaper;
    MoveL Offs(pOrigin,317.42,110.13,0.00),v40,z0,tPen\WObj:=wPaper;
    MoveL Offs(pOrigin,317.97,109.39,0.00),v40,z0,tPen\WObj:=wPaper;
    MoveL Offs(pOrigin,316.02,111.34,0.00),v40,z0,tPen\WObj:=wPaper;
    MoveL Offs(pOrigin,315.18,110.87,0.00),v40,z0,tPen\WObj:=wPaper;
    MoveL Offs(pOrigin,313.37,109.07,0.00),v40,z0,tPen\WObj:=wPaper;
    MoveL Offs(pOrigin,313.03,108.36,0.00),v40,z0,tPen\WObj:=wPaper;
    MoveL Offs(pOrigin,311.08,110.31,0.00),v40,z0,tPen\WObj:=wPaper;
    MoveL Offs(pOrigin,311.13,109.81,0.00),v40,z0,tPen\WObj:=wPaper;
    MoveL Offs(pOrigin,309.33,108.01,0.00),v40,z0,tPen\WObj:=wPaper;
    MoveL Offs(pOrigin,309.44,107.47,0.00),v40,z0,tPen\WObj:=wPaper;
    MoveL Offs(pOrigin,307.49,109.42,0.00),v40,z0,tPen\WObj:=wPaper;
    MoveL Offs(pOrigin,307.08,108.75,0.00),v40,z0,tPen\WObj:=wPaper;
    MoveL Offs(pOrigin,305.58,107.25,0.00),v40,z0,tPen\WObj:=wPaper;
    MoveL Offs(pOrigin,305.85,106.58,0.00),v40,z0,tPen\WObj:=wPaper;
    MoveL Offs(pOrigin,303.89,108.54,0.00),v40,z0,tPen\WObj:=wPaper;
    MoveL Offs(pOrigin,303.18,107.84,0.00),v40,z0,tPen\WObj:=wPaper;
    MoveL Offs(pOrigin,301.68,106.34,0.00),v40,z0,tPen\WObj:=wPaper;
    MoveL Offs(pOrigin,302.26,105.69,0.00),v40,z0,tPen\WObj:=wPaper;
    MoveL Offs(pOrigin,300.30,107.65,0.00),v40,z0,tPen\WObj:=wPaper;
    MoveL Offs(pOrigin,299.59,107.23,0.00),v40,z0,tPen\WObj:=wPaper;
    MoveL Offs(pOrigin,297.93,105.58,0.00),v40,z0,tPen\WObj:=wPaper;
    MoveL Offs(pOrigin,298.51,104.96,0.00),v40,z0,tPen\WObj:=wPaper;
    MoveL Offs(pOrigin,293.55,109.92,0.00),v40,z0,tPen\WObj:=wPaper;
    MoveL Offs(pOrigin,294.20,108.98,0.00),v40,z0,tPen\WObj:=wPaper;
    MoveL Offs(pOrigin,295.26,108.98,0.00),v40,z0,tPen\WObj:=wPaper;
    MoveL Offs(pOrigin,296.25,108.71,0.00),v40,z0,tPen\WObj:=wPaper;
    MoveL Offs(pOrigin,293.70,111.26,0.00),v40,z0,tPen\WObj:=wPaper;
    MoveL Offs(pOrigin,294.15,112.31,0.00),v40,z0,tPen\WObj:=wPaper;
    MoveL Offs(pOrigin,296.55,109.91,0.00),v40,fine,tPen\WObj:=wPaper;
    MoveL Offs(pOrigin,296.55,109.91,6.00),v60,z5,tPen\WObj:=wPaper;
    MoveL Offs(pOrigin,297.76,107.21,6.00),vTravel,z5,tPen\WObj:=wPaper;
    MoveL Offs(pOrigin,297.76,107.21,0.00),v60,z0,tPen\WObj:=wPaper;
    MoveL Offs(pOrigin,299.71,105.25,0.00),v40,z0,tPen\WObj:=wPaper;
    MoveL Offs(pOrigin,299.58,105.73,0.00),v40,z0,tPen\WObj:=wPaper;
    MoveL Offs(pOrigin,301.24,107.39,0.00),v40,z0,tPen\WObj:=wPaper;
  ENDPROC

  PROC DrawPart137()
    MoveL Offs(pOrigin,301.35,108.09,0.00),v40,z0,tPen\WObj:=wPaper;
    MoveL Offs(pOrigin,303.30,106.14,0.00),v40,z0,tPen\WObj:=wPaper;
    MoveL Offs(pOrigin,303.33,106.49,0.00),v40,z0,tPen\WObj:=wPaper;
    MoveL Offs(pOrigin,305.13,108.30,0.00),v40,z0,tPen\WObj:=wPaper;
    MoveL Offs(pOrigin,305.09,108.83,0.00),v40,z0,tPen\WObj:=wPaper;
    MoveL Offs(pOrigin,307.05,106.88,0.00),v40,z0,tPen\WObj:=wPaper;
    MoveL Offs(pOrigin,307.38,107.55,0.00),v40,z0,tPen\WObj:=wPaper;
    MoveL Offs(pOrigin,309.18,109.36,0.00),v40,z0,tPen\WObj:=wPaper;
    MoveL Offs(pOrigin,308.68,109.72,0.00),v40,z0,tPen\WObj:=wPaper;
    MoveL Offs(pOrigin,310.64,107.77,0.00),v40,z0,tPen\WObj:=wPaper;
    MoveL Offs(pOrigin,311.28,108.47,0.00),v40,z0,tPen\WObj:=wPaper;
    MoveL Offs(pOrigin,313.08,110.27,0.00),v40,z0,tPen\WObj:=wPaper;
    MoveL Offs(pOrigin,313.62,110.75,0.00),v40,z0,tPen\WObj:=wPaper;
    MoveL Offs(pOrigin,315.43,108.95,0.00),v40,z0,tPen\WObj:=wPaper;
    MoveL Offs(pOrigin,315.32,109.53,0.00),v40,z0,tPen\WObj:=wPaper;
    MoveL Offs(pOrigin,317.13,111.33,0.00),v40,z0,tPen\WObj:=wPaper;
    MoveL Offs(pOrigin,317.07,111.79,0.00),v40,z0,tPen\WObj:=wPaper;
    MoveL Offs(pOrigin,319.02,109.84,0.00),v40,z0,tPen\WObj:=wPaper;
    MoveL Offs(pOrigin,319.37,110.59,0.00),v40,z0,tPen\WObj:=wPaper;
    MoveL Offs(pOrigin,321.17,112.39,0.00),v40,z0,tPen\WObj:=wPaper;
    MoveL Offs(pOrigin,320.66,112.68,0.00),v40,z0,tPen\WObj:=wPaper;
    MoveL Offs(pOrigin,322.61,110.73,0.00),v40,z0,tPen\WObj:=wPaper;
    MoveL Offs(pOrigin,323.66,111.17,0.00),v40,z0,tPen\WObj:=wPaper;
    MoveL Offs(pOrigin,321.71,113.12,0.00),v40,fine,tPen\WObj:=wPaper;
    MoveL Offs(pOrigin,321.71,113.12,6.00),v60,z5,tPen\WObj:=wPaper;
    MoveL Offs(pOrigin,323.05,113.27,6.00),vTravel,z5,tPen\WObj:=wPaper;
    MoveL Offs(pOrigin,323.05,113.27,0.00),v60,z0,tPen\WObj:=wPaper;
    MoveL Offs(pOrigin,325.01,111.32,0.00),v40,fine,tPen\WObj:=wPaper;
    MoveL Offs(pOrigin,325.01,111.32,6.00),v60,z5,tPen\WObj:=wPaper;
    MoveL Offs(pOrigin,323.42,111.65,6.00),vTravel,z5,tPen\WObj:=wPaper;
    MoveL Offs(pOrigin,323.42,111.65,0.00),v60,z0,tPen\WObj:=wPaper;
    MoveL Offs(pOrigin,325.37,113.60,0.00),v40,z0,tPen\WObj:=wPaper;
    MoveL Offs(pOrigin,325.45,113.86,0.00),v40,z0,tPen\WObj:=wPaper;
    MoveL Offs(pOrigin,327.40,111.91,0.00),v40,z0,tPen\WObj:=wPaper;
    MoveL Offs(pOrigin,327.47,112.71,0.00),v40,z0,tPen\WObj:=wPaper;
    MoveL Offs(pOrigin,329.57,114.81,0.00),v40,z0,tPen\WObj:=wPaper;
    MoveL Offs(pOrigin,329.94,115.35,0.00),v40,z0,tPen\WObj:=wPaper;
    MoveL Offs(pOrigin,331.89,113.39,0.00),v40,z0,tPen\WObj:=wPaper;
    MoveL Offs(pOrigin,331.51,113.77,0.00),v40,z0,tPen\WObj:=wPaper;
    MoveL Offs(pOrigin,333.77,116.02,0.00),v40,z0,tPen\WObj:=wPaper;
    MoveL Offs(pOrigin,333.38,116.38,0.00),v40,z0,tPen\WObj:=wPaper;
    MoveL Offs(pOrigin,335.33,114.43,0.00),v40,z0,tPen\WObj:=wPaper;
    MoveL Offs(pOrigin,335.86,115.13,0.00),v40,z0,tPen\WObj:=wPaper;
    MoveL Offs(pOrigin,338.12,117.39,0.00),v40,z0,tPen\WObj:=wPaper;
    MoveL Offs(pOrigin,338.17,117.57,0.00),v40,z0,tPen\WObj:=wPaper;
    MoveL Offs(pOrigin,340.12,115.62,0.00),v40,z0,tPen\WObj:=wPaper;
    MoveL Offs(pOrigin,340.06,116.34,0.00),v40,z0,tPen\WObj:=wPaper;
    MoveL Offs(pOrigin,342.32,118.60,0.00),v40,z0,tPen\WObj:=wPaper;
    MoveL Offs(pOrigin,342.66,119.05,0.00),v40,z0,tPen\WObj:=wPaper;
    MoveL Offs(pOrigin,344.61,117.10,0.00),v40,z0,tPen\WObj:=wPaper;
    MoveL Offs(pOrigin,344.56,117.85,0.00),v40,z0,tPen\WObj:=wPaper;
    MoveL Offs(pOrigin,345.61,118.91,0.00),v40,z0,tPen\WObj:=wPaper;
    MoveL Offs(pOrigin,345.96,118.74,0.00),v40,z0,tPen\WObj:=wPaper;
    MoveL Offs(pOrigin,343.85,120.85,0.00),v40,z0,tPen\WObj:=wPaper;
    MoveL Offs(pOrigin,344.27,120.55,0.00),v40,z0,tPen\WObj:=wPaper;
    MoveL Offs(pOrigin,345.92,122.20,0.00),v40,z0,tPen\WObj:=wPaper;
    MoveL Offs(pOrigin,346.39,122.79,0.00),v40,z0,tPen\WObj:=wPaper;
    MoveL Offs(pOrigin,343.84,125.34,0.00),v40,z0,tPen\WObj:=wPaper;
    MoveL Offs(pOrigin,344.43,125.19,0.00),v40,z0,tPen\WObj:=wPaper;
    MoveL Offs(pOrigin,345.94,126.70,0.00),v40,z0,tPen\WObj:=wPaper;
    MoveL Offs(pOrigin,346.38,127.28,0.00),v40,z0,tPen\WObj:=wPaper;
    MoveL Offs(pOrigin,342.92,130.74,0.00),v40,z0,tPen\WObj:=wPaper;
    MoveL Offs(pOrigin,343.70,130.44,0.00),v40,z0,tPen\WObj:=wPaper;
    MoveL Offs(pOrigin,341.30,128.03,0.00),v40,z0,tPen\WObj:=wPaper;
    MoveL Offs(pOrigin,341.89,127.29,0.00),v40,z0,tPen\WObj:=wPaper;
    MoveL Offs(pOrigin,337.23,131.95,0.00),v40,z0,tPen\WObj:=wPaper;
    MoveL Offs(pOrigin,338.12,132.55,0.00),v40,z0,tPen\WObj:=wPaper;
    MoveL Offs(pOrigin,339.63,131.05,0.00),v40,z0,tPen\WObj:=wPaper;
    MoveL Offs(pOrigin,340.37,131.79,0.00),v40,z0,tPen\WObj:=wPaper;
    MoveL Offs(pOrigin,338.87,133.30,0.00),v40,z0,tPen\WObj:=wPaper;
    MoveL Offs(pOrigin,339.77,133.89,0.00),v40,z0,tPen\WObj:=wPaper;
    MoveL Offs(pOrigin,341.27,132.39,0.00),v40,z0,tPen\WObj:=wPaper;
    MoveL Offs(pOrigin,342.17,132.99,0.00),v40,z0,tPen\WObj:=wPaper;
    MoveL Offs(pOrigin,340.51,134.64,0.00),v40,z0,tPen\WObj:=wPaper;
    MoveL Offs(pOrigin,341.41,135.23,0.00),v40,z0,tPen\WObj:=wPaper;
    MoveL Offs(pOrigin,343.06,133.58,0.00),v40,fine,tPen\WObj:=wPaper;
    MoveL Offs(pOrigin,343.06,133.58,6.00),v60,z5,tPen\WObj:=wPaper;
    MoveL Offs(pOrigin,342.23,134.62,6.00),vTravel,z5,tPen\WObj:=wPaper;
    MoveL Offs(pOrigin,342.23,134.62,0.00),v60,z0,tPen\WObj:=wPaper;
    MoveL Offs(pOrigin,342.65,134.84,0.00),v40,z0,tPen\WObj:=wPaper;
    MoveL Offs(pOrigin,342.23,134.62,0.00),v40,fine,tPen\WObj:=wPaper;
    MoveL Offs(pOrigin,342.23,134.62,6.00),v60,z5,tPen\WObj:=wPaper;
    MoveL Offs(pOrigin,344.27,130.88,6.00),vTravel,z5,tPen\WObj:=wPaper;
    MoveL Offs(pOrigin,344.27,130.88,0.00),v60,z0,tPen\WObj:=wPaper;
    MoveL Offs(pOrigin,346.22,128.93,0.00),v40,z0,tPen\WObj:=wPaper;
    MoveL Offs(pOrigin,345.64,129.39,0.00),v40,z0,tPen\WObj:=wPaper;
    MoveL Offs(pOrigin,344.14,127.89,0.00),v40,z0,tPen\WObj:=wPaper;
    MoveL Offs(pOrigin,343.24,128.49,0.00),v40,z0,tPen\WObj:=wPaper;
    MoveL Offs(pOrigin,345.05,130.29,0.00),v40,z0,tPen\WObj:=wPaper;
    MoveL Offs(pOrigin,344.99,130.38,0.00),v40,z0,tPen\WObj:=wPaper;
    MoveL Offs(pOrigin,345.20,129.95,0.00),v40,z0,tPen\WObj:=wPaper;
    MoveL Offs(pOrigin,344.99,130.38,0.00),v40,fine,tPen\WObj:=wPaper;
    MoveL Offs(pOrigin,344.99,130.38,6.00),v60,z5,tPen\WObj:=wPaper;
    MoveL Offs(pOrigin,345.20,129.05,6.00),vTravel,z5,tPen\WObj:=wPaper;
    MoveL Offs(pOrigin,345.20,129.05,0.00),v60,z0,tPen\WObj:=wPaper;
    MoveL Offs(pOrigin,343.50,129.05,0.00),v40,fine,tPen\WObj:=wPaper;
    MoveL Offs(pOrigin,343.50,129.05,6.00),v60,z5,tPen\WObj:=wPaper;
    MoveL Offs(pOrigin,341.88,130.29,6.00),vTravel,z5,tPen\WObj:=wPaper;
    MoveL Offs(pOrigin,341.88,130.29,0.00),v60,z0,tPen\WObj:=wPaper;
    MoveL Offs(pOrigin,346.38,125.78,0.00),v40,z0,tPen\WObj:=wPaper;
    MoveL Offs(pOrigin,345.93,125.20,0.00),v40,z0,tPen\WObj:=wPaper;
    MoveL Offs(pOrigin,344.43,123.70,0.00),v40,z0,tPen\WObj:=wPaper;
    MoveL Offs(pOrigin,343.84,123.84,0.00),v40,z0,tPen\WObj:=wPaper;
    MoveL Offs(pOrigin,346.40,121.29,0.00),v40,fine,tPen\WObj:=wPaper;
    MoveL Offs(pOrigin,346.40,121.29,6.00),v60,z5,tPen\WObj:=wPaper;
    MoveL Offs(pOrigin,349.10,120.08,6.00),vTravel,z5,tPen\WObj:=wPaper;
    MoveL Offs(pOrigin,349.10,120.08,0.00),v60,z0,tPen\WObj:=wPaper;
    MoveL Offs(pOrigin,354.66,114.52,0.00),v40,z0,tPen\WObj:=wPaper;
    MoveL Offs(pOrigin,355.40,115.27,0.00),v40,z0,tPen\WObj:=wPaper;
    MoveL Offs(pOrigin,353.45,117.22,0.00),v40,z0,tPen\WObj:=wPaper;
    MoveL Offs(pOrigin,354.05,118.12,0.00),v40,z0,tPen\WObj:=wPaper;
    MoveL Offs(pOrigin,356.00,116.17,0.00),v40,z0,tPen\WObj:=wPaper;
    MoveL Offs(pOrigin,356.60,117.06,0.00),v40,z0,tPen\WObj:=wPaper;
    MoveL Offs(pOrigin,354.79,118.87,0.00),v40,fine,tPen\WObj:=wPaper;
    MoveL Offs(pOrigin,354.79,118.87,6.00),v60,z5,tPen\WObj:=wPaper;
    MoveL Offs(pOrigin,355.40,117.41,6.00),vTravel,z5,tPen\WObj:=wPaper;
    MoveL Offs(pOrigin,355.40,117.41,0.00),v60,z0,tPen\WObj:=wPaper;
    MoveL Offs(pOrigin,355.19,116.35,0.00),v40,z0,tPen\WObj:=wPaper;
    MoveL Offs(pOrigin,354.55,116.35,0.00),v40,z0,tPen\WObj:=wPaper;
    MoveL Offs(pOrigin,354.55,116.35,0.00),v40,z0,tPen\WObj:=wPaper;
  ENDPROC

  PROC DrawPart138()
    MoveL Offs(pOrigin,354.34,115.50,0.00),v40,z0,tPen\WObj:=wPaper;
    MoveL Offs(pOrigin,353.49,115.29,0.00),v40,z0,tPen\WObj:=wPaper;
    MoveL Offs(pOrigin,353.49,115.29,0.00),v40,z0,tPen\WObj:=wPaper;
    MoveL Offs(pOrigin,350.80,111.04,0.00),v40,z0,tPen\WObj:=wPaper;
    MoveL Offs(pOrigin,351.15,110.26,0.00),v40,z0,tPen\WObj:=wPaper;
    MoveL Offs(pOrigin,352.42,110.54,0.00),v40,z0,tPen\WObj:=wPaper;
    MoveL Offs(pOrigin,356.46,113.45,0.00),v40,z0,tPen\WObj:=wPaper;
    MoveL Offs(pOrigin,358.59,114.44,0.00),v40,z0,tPen\WObj:=wPaper;
    MoveL Offs(pOrigin,358.59,114.44,0.00),v40,z0,tPen\WObj:=wPaper;
    MoveL Offs(pOrigin,358.80,114.86,0.00),v40,z0,tPen\WObj:=wPaper;
    MoveL Offs(pOrigin,359.44,115.07,0.00),v40,z0,tPen\WObj:=wPaper;
    MoveL Offs(pOrigin,359.86,114.86,0.00),v40,z0,tPen\WObj:=wPaper;
    MoveL Offs(pOrigin,359.86,114.86,0.00),v40,z0,tPen\WObj:=wPaper;
    MoveL Offs(pOrigin,359.44,114.01,0.00),v40,z0,tPen\WObj:=wPaper;
    MoveL Offs(pOrigin,358.59,114.01,0.00),v40,z0,tPen\WObj:=wPaper;
    MoveL Offs(pOrigin,358.59,114.01,0.00),v40,z0,tPen\WObj:=wPaper;
    MoveL Offs(pOrigin,358.38,113.45,0.00),v40,z0,tPen\WObj:=wPaper;
    MoveL Offs(pOrigin,354.12,110.40,0.00),v40,z0,tPen\WObj:=wPaper;
    MoveL Offs(pOrigin,351.15,107.43,0.00),v40,z0,tPen\WObj:=wPaper;
    MoveL Offs(pOrigin,350.02,105.72,0.00),v40,z0,tPen\WObj:=wPaper;
    MoveL Offs(pOrigin,349.45,104.03,0.00),v40,z0,tPen\WObj:=wPaper;
    MoveL Offs(pOrigin,349.52,102.96,0.00),v40,z0,tPen\WObj:=wPaper;
    MoveL Offs(pOrigin,350.51,103.18,0.00),v40,z0,tPen\WObj:=wPaper;
    MoveL Offs(pOrigin,352.64,105.30,0.00),v40,z0,tPen\WObj:=wPaper;
    MoveL Offs(pOrigin,356.67,108.28,0.00),v40,z0,tPen\WObj:=wPaper;
    MoveL Offs(pOrigin,356.67,108.28,0.00),v40,z0,tPen\WObj:=wPaper;
    MoveL Offs(pOrigin,357.52,109.12,0.00),v40,z0,tPen\WObj:=wPaper;
    MoveL Offs(pOrigin,358.59,109.34,0.00),v40,z0,tPen\WObj:=wPaper;
    MoveL Offs(pOrigin,357.67,110.02,0.00),v40,z0,tPen\WObj:=wPaper;
    MoveL Offs(pOrigin,359.47,108.22,0.00),v40,z0,tPen\WObj:=wPaper;
    MoveL Offs(pOrigin,358.61,108.01,0.00),v40,z0,tPen\WObj:=wPaper;
    MoveL Offs(pOrigin,363.87,113.27,0.00),v40,z0,tPen\WObj:=wPaper;
    MoveL Offs(pOrigin,363.35,113.30,0.00),v40,z0,tPen\WObj:=wPaper;
    MoveL Offs(pOrigin,365.15,111.49,0.00),v40,z0,tPen\WObj:=wPaper;
    MoveL Offs(pOrigin,365.90,112.24,0.00),v40,z0,tPen\WObj:=wPaper;
    MoveL Offs(pOrigin,364.25,113.89,0.00),v40,z0,tPen\WObj:=wPaper;
    MoveL Offs(pOrigin,364.99,114.64,0.00),v40,z0,tPen\WObj:=wPaper;
    MoveL Offs(pOrigin,366.95,112.69,0.00),v40,z0,tPen\WObj:=wPaper;
    MoveL Offs(pOrigin,366.72,113.13,0.00),v40,z0,tPen\WObj:=wPaper;
    MoveL Offs(pOrigin,370.17,116.59,0.00),v40,z0,tPen\WObj:=wPaper;
    MoveL Offs(pOrigin,369.93,117.17,0.00),v40,z0,tPen\WObj:=wPaper;
    MoveL Offs(pOrigin,371.88,115.22,0.00),v40,fine,tPen\WObj:=wPaper;
    MoveL Offs(pOrigin,371.88,115.22,6.00),v60,z5,tPen\WObj:=wPaper;
    MoveL Offs(pOrigin,369.64,118.47,6.00),vTravel,z5,tPen\WObj:=wPaper;
    MoveL Offs(pOrigin,369.64,118.47,0.00),v60,z0,tPen\WObj:=wPaper;
    MoveL Offs(pOrigin,369.21,118.62,0.00),v40,z0,tPen\WObj:=wPaper;
    MoveL Offs(pOrigin,365.39,117.34,0.00),v40,z0,tPen\WObj:=wPaper;
    MoveL Offs(pOrigin,359.86,114.86,0.00),v40,z0,tPen\WObj:=wPaper;
    MoveL Offs(pOrigin,359.30,115.86,0.00),v40,z0,tPen\WObj:=wPaper;
    MoveL Offs(pOrigin,361.10,114.05,0.00),v40,z0,tPen\WObj:=wPaper;
    MoveL Offs(pOrigin,360.20,113.46,0.00),v40,z0,tPen\WObj:=wPaper;
    MoveL Offs(pOrigin,358.25,115.41,0.00),v40,fine,tPen\WObj:=wPaper;
    MoveL Offs(pOrigin,358.25,115.41,6.00),v60,z5,tPen\WObj:=wPaper;
    MoveL Offs(pOrigin,358.16,113.21,6.00),vTravel,z5,tPen\WObj:=wPaper;
    MoveL Offs(pOrigin,358.16,113.21,0.00),v60,z0,tPen\WObj:=wPaper;
    MoveL Offs(pOrigin,356.67,113.21,0.00),v40,fine,tPen\WObj:=wPaper;
    MoveL Offs(pOrigin,356.67,113.21,6.00),v60,z5,tPen\WObj:=wPaper;
    MoveL Offs(pOrigin,356.31,114.37,6.00),vTravel,z5,tPen\WObj:=wPaper;
    MoveL Offs(pOrigin,356.31,114.37,0.00),v60,z0,tPen\WObj:=wPaper;
    MoveL Offs(pOrigin,358.41,112.26,0.00),v40,fine,tPen\WObj:=wPaper;
    MoveL Offs(pOrigin,358.41,112.26,6.00),v60,z5,tPen\WObj:=wPaper;
    MoveL Offs(pOrigin,359.46,111.21,6.00),vTravel,z5,tPen\WObj:=wPaper;
    MoveL Offs(pOrigin,359.46,111.21,0.00),v60,z0,tPen\WObj:=wPaper;
    MoveL Offs(pOrigin,361.26,109.41,0.00),v40,z0,tPen\WObj:=wPaper;
    MoveL Offs(pOrigin,360.37,108.81,0.00),v40,z0,tPen\WObj:=wPaper;
    MoveL Offs(pOrigin,358.56,110.62,0.00),v40,fine,tPen\WObj:=wPaper;
    MoveL Offs(pOrigin,358.56,110.62,6.00),v60,z5,tPen\WObj:=wPaper;
    MoveL Offs(pOrigin,356.62,111.07,6.00),vTravel,z5,tPen\WObj:=wPaper;
    MoveL Offs(pOrigin,356.62,111.07,0.00),v60,z0,tPen\WObj:=wPaper;
    MoveL Offs(pOrigin,348.80,118.88,0.00),v40,z0,tPen\WObj:=wPaper;
    MoveL Offs(pOrigin,349.66,118.49,0.00),v40,z0,tPen\WObj:=wPaper;
    MoveL Offs(pOrigin,352.00,118.49,0.00),v40,z0,tPen\WObj:=wPaper;
    MoveL Offs(pOrigin,352.55,118.12,0.00),v40,z0,tPen\WObj:=wPaper;
    MoveL Offs(pOrigin,349.39,121.28,0.00),v40,z0,tPen\WObj:=wPaper;
    MoveL Offs(pOrigin,349.66,121.47,0.00),v40,z0,tPen\WObj:=wPaper;
    MoveL Offs(pOrigin,360.48,132.28,0.00),v40,z0,tPen\WObj:=wPaper;
    MoveL Offs(pOrigin,360.08,132.50,0.00),v40,z0,tPen\WObj:=wPaper;
    MoveL Offs(pOrigin,364.75,137.18,0.00),v40,z0,tPen\WObj:=wPaper;
    MoveL Offs(pOrigin,360.08,132.50,0.00),v40,z0,tPen\WObj:=wPaper;
    MoveL Offs(pOrigin,361.05,132.03,0.00),v40,z0,tPen\WObj:=wPaper;
    MoveL Offs(pOrigin,356.84,136.24,0.00),v40,z0,tPen\WObj:=wPaper;
    MoveL Offs(pOrigin,357.58,136.98,0.00),v40,z0,tPen\WObj:=wPaper;
    MoveL Offs(pOrigin,361.64,132.93,0.00),v40,z0,tPen\WObj:=wPaper;
    MoveL Offs(pOrigin,360.92,133.27,0.00),v40,z0,tPen\WObj:=wPaper;
    MoveL Offs(pOrigin,359.01,133.27,0.00),v40,z0,tPen\WObj:=wPaper;
    MoveL Offs(pOrigin,359.23,133.35,0.00),v40,z0,tPen\WObj:=wPaper;
    MoveL Offs(pOrigin,360.08,134.20,0.00),v40,z0,tPen\WObj:=wPaper;
    MoveL Offs(pOrigin,359.23,133.35,0.00),v40,fine,tPen\WObj:=wPaper;
    MoveL Offs(pOrigin,359.23,133.35,6.00),v60,z5,tPen\WObj:=wPaper;
    MoveL Offs(pOrigin,360.08,134.33,6.00),vTravel,z5,tPen\WObj:=wPaper;
    MoveL Offs(pOrigin,360.08,134.33,0.00),v60,z0,tPen\WObj:=wPaper;
    MoveL Offs(pOrigin,361.99,134.33,0.00),v40,fine,tPen\WObj:=wPaper;
    MoveL Offs(pOrigin,361.99,134.33,6.00),v60,z5,tPen\WObj:=wPaper;
    MoveL Offs(pOrigin,360.29,134.41,6.00),vTravel,z5,tPen\WObj:=wPaper;
    MoveL Offs(pOrigin,360.29,134.41,0.00),v60,z0,tPen\WObj:=wPaper;
    MoveL Offs(pOrigin,360.71,134.84,0.00),v40,z0,tPen\WObj:=wPaper;
    MoveL Offs(pOrigin,360.29,134.41,0.00),v40,fine,tPen\WObj:=wPaper;
    MoveL Offs(pOrigin,360.29,134.41,6.00),v60,z5,tPen\WObj:=wPaper;
    MoveL Offs(pOrigin,359.01,136.54,6.00),vTravel,z5,tPen\WObj:=wPaper;
    MoveL Offs(pOrigin,359.01,136.54,0.00),v60,z0,tPen\WObj:=wPaper;
    MoveL Offs(pOrigin,358.94,135.90,0.00),v40,z0,tPen\WObj:=wPaper;
    MoveL Offs(pOrigin,356.67,132.93,0.00),v40,z0,tPen\WObj:=wPaper;
    MoveL Offs(pOrigin,355.61,132.50,0.00),v40,fine,tPen\WObj:=wPaper;
    MoveL Offs(pOrigin,355.61,132.50,6.00),v60,z5,tPen\WObj:=wPaper;
    MoveL Offs(pOrigin,355.19,131.16,6.00),vTravel,z5,tPen\WObj:=wPaper;
    MoveL Offs(pOrigin,355.19,131.16,0.00),v60,z0,tPen\WObj:=wPaper;
    MoveL Offs(pOrigin,352.21,131.16,0.00),v40,z0,tPen\WObj:=wPaper;
    MoveL Offs(pOrigin,352.72,130.80,0.00),v40,z0,tPen\WObj:=wPaper;
    MoveL Offs(pOrigin,352.72,127.19,0.00),v40,fine,tPen\WObj:=wPaper;
    MoveL Offs(pOrigin,352.72,127.19,6.00),v60,z5,tPen\WObj:=wPaper;
    MoveL Offs(pOrigin,353.70,125.70,6.00),vTravel,z5,tPen\WObj:=wPaper;
    MoveL Offs(pOrigin,353.70,125.70,0.00),v60,z0,tPen\WObj:=wPaper;
    MoveL Offs(pOrigin,354.12,126.34,0.00),v40,z0,tPen\WObj:=wPaper;
    MoveL Offs(pOrigin,353.70,125.70,0.00),v40,z0,tPen\WObj:=wPaper;
    MoveL Offs(pOrigin,353.77,125.70,0.00),v40,z0,tPen\WObj:=wPaper;
    MoveL Offs(pOrigin,353.77,124.21,0.00),v40,z0,tPen\WObj:=wPaper;
    MoveL Offs(pOrigin,354.34,123.77,0.00),v40,z0,tPen\WObj:=wPaper;
    MoveL Offs(pOrigin,350.72,123.77,0.00),v40,z0,tPen\WObj:=wPaper;
    MoveL Offs(pOrigin,349.97,123.26,0.00),v40,z0,tPen\WObj:=wPaper;
    MoveL Offs(pOrigin,368.00,141.30,0.00),v40,z0,tPen\WObj:=wPaper;
  ENDPROC

  PROC DrawPart139()
    MoveL Offs(pOrigin,367.91,141.59,0.00),v40,z0,tPen\WObj:=wPaper;
    MoveL Offs(pOrigin,369.86,139.64,0.00),v40,z0,tPen\WObj:=wPaper;
    MoveL Offs(pOrigin,368.96,139.05,0.00),v40,z0,tPen\WObj:=wPaper;
    MoveL Offs(pOrigin,367.01,141.00,0.00),v40,z0,tPen\WObj:=wPaper;
    MoveL Offs(pOrigin,365.96,140.55,0.00),v40,z0,tPen\WObj:=wPaper;
    MoveL Offs(pOrigin,368.07,138.45,0.00),v40,z0,tPen\WObj:=wPaper;
    MoveL Offs(pOrigin,367.32,137.70,0.00),v40,z0,tPen\WObj:=wPaper;
    MoveL Offs(pOrigin,360.86,144.16,0.00),v40,z0,tPen\WObj:=wPaper;
    MoveL Offs(pOrigin,361.72,143.97,0.00),v40,z0,tPen\WObj:=wPaper;
    MoveL Offs(pOrigin,369.38,151.64,0.00),v40,z0,tPen\WObj:=wPaper;
    MoveL Offs(pOrigin,369.97,151.48,0.00),v40,z0,tPen\WObj:=wPaper;
    MoveL Offs(pOrigin,367.87,153.58,0.00),v40,z0,tPen\WObj:=wPaper;
    MoveL Offs(pOrigin,368.04,153.28,0.00),v40,z0,tPen\WObj:=wPaper;
    MoveL Offs(pOrigin,381.11,166.35,0.00),v40,z0,tPen\WObj:=wPaper;
    MoveL Offs(pOrigin,380.69,166.01,0.00),v40,z0,tPen\WObj:=wPaper;
    MoveL Offs(pOrigin,378.56,166.01,0.00),v40,z0,tPen\WObj:=wPaper;
    MoveL Offs(pOrigin,378.26,166.49,0.00),v40,z0,tPen\WObj:=wPaper;
    MoveL Offs(pOrigin,381.87,170.10,0.00),v40,z0,tPen\WObj:=wPaper;
    MoveL Offs(pOrigin,381.54,170.23,0.00),v40,z0,tPen\WObj:=wPaper;
    MoveL Offs(pOrigin,380.48,170.23,0.00),v40,z0,tPen\WObj:=wPaper;
    MoveL Offs(pOrigin,380.26,171.29,0.00),v40,z0,tPen\WObj:=wPaper;
    MoveL Offs(pOrigin,381.33,171.29,0.00),v40,z0,tPen\WObj:=wPaper;
    MoveL Offs(pOrigin,381.72,171.45,0.00),v40,z0,tPen\WObj:=wPaper;
    MoveL Offs(pOrigin,379.47,169.19,0.00),v40,z0,tPen\WObj:=wPaper;
    MoveL Offs(pOrigin,379.21,169.12,0.00),v40,z0,tPen\WObj:=wPaper;
    MoveL Offs(pOrigin,381.76,166.57,0.00),v40,z0,tPen\WObj:=wPaper;
    MoveL Offs(pOrigin,380.90,167.06,0.00),v40,z0,tPen\WObj:=wPaper;
    MoveL Offs(pOrigin,379.41,167.06,0.00),v40,z0,tPen\WObj:=wPaper;
    MoveL Offs(pOrigin,378.77,166.71,0.00),v40,z0,tPen\WObj:=wPaper;
    MoveL Offs(pOrigin,378.99,167.14,0.00),v40,z0,tPen\WObj:=wPaper;
    MoveL Offs(pOrigin,378.77,166.71,0.00),v40,z0,tPen\WObj:=wPaper;
    MoveL Offs(pOrigin,379.12,166.29,0.00),v40,z0,tPen\WObj:=wPaper;
    MoveL Offs(pOrigin,379.12,164.16,0.00),v40,z0,tPen\WObj:=wPaper;
    MoveL Offs(pOrigin,380.17,163.74,0.00),v40,z0,tPen\WObj:=wPaper;
    MoveL Offs(pOrigin,380.17,167.56,0.00),v40,z0,tPen\WObj:=wPaper;
    MoveL Offs(pOrigin,379.84,168.12,0.00),v40,z0,tPen\WObj:=wPaper;
    MoveL Offs(pOrigin,381.11,168.12,0.00),v40,z0,tPen\WObj:=wPaper;
    MoveL Offs(pOrigin,381.33,169.18,0.00),v40,z0,tPen\WObj:=wPaper;
    MoveL Offs(pOrigin,380.26,169.18,0.00),v40,fine,tPen\WObj:=wPaper;
    MoveL Offs(pOrigin,380.26,169.18,6.00),v60,z5,tPen\WObj:=wPaper;
    MoveL Offs(pOrigin,378.76,168.08,6.00),vTravel,z5,tPen\WObj:=wPaper;
    MoveL Offs(pOrigin,378.76,168.08,0.00),v60,z0,tPen\WObj:=wPaper;
    MoveL Offs(pOrigin,381.77,165.07,0.00),v40,z0,tPen\WObj:=wPaper;
    MoveL Offs(pOrigin,381.11,164.85,0.00),v40,z0,tPen\WObj:=wPaper;
    MoveL Offs(pOrigin,379.15,162.90,0.00),v40,z0,tPen\WObj:=wPaper;
    MoveL Offs(pOrigin,379.84,162.84,0.00),v40,z0,tPen\WObj:=wPaper;
    MoveL Offs(pOrigin,381.11,162.84,0.00),v40,z0,tPen\WObj:=wPaper;
    MoveL Offs(pOrigin,381.85,162.61,0.00),v40,z0,tPen\WObj:=wPaper;
    MoveL Offs(pOrigin,380.19,160.96,0.00),v40,z0,tPen\WObj:=wPaper;
    MoveL Offs(pOrigin,380.69,160.73,0.00),v40,z0,tPen\WObj:=wPaper;
    MoveL Offs(pOrigin,381.96,160.73,0.00),v40,z0,tPen\WObj:=wPaper;
    MoveL Offs(pOrigin,382.14,161.41,0.00),v40,z0,tPen\WObj:=wPaper;
    MoveL Offs(pOrigin,380.64,159.91,0.00),v40,z0,tPen\WObj:=wPaper;
    MoveL Offs(pOrigin,381.11,159.67,0.00),v40,z0,tPen\WObj:=wPaper;
    MoveL Offs(pOrigin,382.39,159.67,0.00),v40,z0,tPen\WObj:=wPaper;
    MoveL Offs(pOrigin,382.59,160.36,0.00),v40,z0,tPen\WObj:=wPaper;
    MoveL Offs(pOrigin,380.94,158.71,0.00),v40,z0,tPen\WObj:=wPaper;
    MoveL Offs(pOrigin,381.75,158.62,0.00),v40,z0,tPen\WObj:=wPaper;
    MoveL Offs(pOrigin,382.81,158.62,0.00),v40,z0,tPen\WObj:=wPaper;
    MoveL Offs(pOrigin,383.02,158.64,0.00),v40,z0,tPen\WObj:=wPaper;
    MoveL Offs(pOrigin,382.81,159.06,0.00),v40,z0,tPen\WObj:=wPaper;
    MoveL Offs(pOrigin,383.02,158.64,0.00),v40,z0,tPen\WObj:=wPaper;
    MoveL Offs(pOrigin,383.48,158.27,0.00),v40,z0,tPen\WObj:=wPaper;
    MoveL Offs(pOrigin,381.98,156.77,0.00),v40,z0,tPen\WObj:=wPaper;
    MoveL Offs(pOrigin,382.39,156.30,0.00),v40,z0,tPen\WObj:=wPaper;
    MoveL Offs(pOrigin,382.17,156.73,0.00),v40,z0,tPen\WObj:=wPaper;
    MoveL Offs(pOrigin,382.39,156.30,0.00),v40,z0,tPen\WObj:=wPaper;
    MoveL Offs(pOrigin,382.60,156.50,0.00),v40,z0,tPen\WObj:=wPaper;
    MoveL Offs(pOrigin,383.88,156.50,0.00),v40,z0,tPen\WObj:=wPaper;
    MoveL Offs(pOrigin,384.37,156.18,0.00),v40,z0,tPen\WObj:=wPaper;
    MoveL Offs(pOrigin,382.87,154.67,0.00),v40,z0,tPen\WObj:=wPaper;
    MoveL Offs(pOrigin,383.24,154.60,0.00),v40,z0,tPen\WObj:=wPaper;
    MoveL Offs(pOrigin,383.02,155.02,0.00),v40,z0,tPen\WObj:=wPaper;
    MoveL Offs(pOrigin,383.24,154.60,0.00),v40,z0,tPen\WObj:=wPaper;
    MoveL Offs(pOrigin,383.66,154.39,0.00),v40,z0,tPen\WObj:=wPaper;
    MoveL Offs(pOrigin,384.72,154.39,0.00),v40,z0,tPen\WObj:=wPaper;
    MoveL Offs(pOrigin,385.42,154.23,0.00),v40,z0,tPen\WObj:=wPaper;
    MoveL Offs(pOrigin,383.91,152.73,0.00),v40,z0,tPen\WObj:=wPaper;
    MoveL Offs(pOrigin,383.88,153.11,0.00),v40,z0,tPen\WObj:=wPaper;
    MoveL Offs(pOrigin,383.66,153.54,0.00),v40,z0,tPen\WObj:=wPaper;
    MoveL Offs(pOrigin,383.88,153.11,0.00),v40,z0,tPen\WObj:=wPaper;
    MoveL Offs(pOrigin,384.09,153.34,0.00),v40,z0,tPen\WObj:=wPaper;
    MoveL Offs(pOrigin,385.36,153.34,0.00),v40,z0,tPen\WObj:=wPaper;
    MoveL Offs(pOrigin,385.58,153.32,0.00),v40,z0,tPen\WObj:=wPaper;
    MoveL Offs(pOrigin,385.36,153.75,0.00),v40,z0,tPen\WObj:=wPaper;
    MoveL Offs(pOrigin,385.58,153.32,0.00),v40,z0,tPen\WObj:=wPaper;
    MoveL Offs(pOrigin,385.86,153.18,0.00),v40,z0,tPen\WObj:=wPaper;
    MoveL Offs(pOrigin,384.36,151.68,0.00),v40,z0,tPen\WObj:=wPaper;
    MoveL Offs(pOrigin,384.51,152.28,0.00),v40,z0,tPen\WObj:=wPaper;
    MoveL Offs(pOrigin,385.79,152.28,0.00),v40,z0,tPen\WObj:=wPaper;
    MoveL Offs(pOrigin,386.31,152.14,0.00),v40,z0,tPen\WObj:=wPaper;
    MoveL Offs(pOrigin,384.66,150.48,0.00),v40,z0,tPen\WObj:=wPaper;
    MoveL Offs(pOrigin,385.36,150.17,0.00),v40,z0,tPen\WObj:=wPaper;
    MoveL Offs(pOrigin,386.64,150.17,0.00),v40,z0,tPen\WObj:=wPaper;
    MoveL Offs(pOrigin,387.20,150.04,0.00),v40,z0,tPen\WObj:=wPaper;
    MoveL Offs(pOrigin,384.95,147.79,0.00),v40,z0,tPen\WObj:=wPaper;
    MoveL Offs(pOrigin,384.52,147.39,0.00),v40,z0,tPen\WObj:=wPaper;
    MoveL Offs(pOrigin,393.98,137.92,0.00),v40,z0,tPen\WObj:=wPaper;
    MoveL Offs(pOrigin,393.61,138.53,0.00),v40,z0,tPen\WObj:=wPaper;
    MoveL Offs(pOrigin,388.95,133.87,0.00),v40,z0,tPen\WObj:=wPaper;
    MoveL Offs(pOrigin,389.40,134.33,0.00),v40,z0,tPen\WObj:=wPaper;
    MoveL Offs(pOrigin,390.67,134.33,0.00),v40,z0,tPen\WObj:=wPaper;
    MoveL Offs(pOrigin,390.67,135.38,0.00),v40,z0,tPen\WObj:=wPaper;
    MoveL Offs(pOrigin,389.40,135.38,0.00),v40,z0,tPen\WObj:=wPaper;
    MoveL Offs(pOrigin,389.19,136.44,0.00),v40,z0,tPen\WObj:=wPaper;
    MoveL Offs(pOrigin,390.67,136.44,0.00),v40,z0,tPen\WObj:=wPaper;
    MoveL Offs(pOrigin,390.67,137.50,0.00),v40,z0,tPen\WObj:=wPaper;
    MoveL Offs(pOrigin,389.19,137.50,0.00),v40,z0,tPen\WObj:=wPaper;
    MoveL Offs(pOrigin,388.66,138.06,0.00),v40,z0,tPen\WObj:=wPaper;
    MoveL Offs(pOrigin,393.17,142.57,0.00),v40,z0,tPen\WObj:=wPaper;
    MoveL Offs(pOrigin,393.52,142.86,0.00),v40,z0,tPen\WObj:=wPaper;
    MoveL Offs(pOrigin,389.91,146.47,0.00),v40,z0,tPen\WObj:=wPaper;
    MoveL Offs(pOrigin,390.63,146.01,0.00),v40,z0,tPen\WObj:=wPaper;
    MoveL Offs(pOrigin,392.59,147.96,0.00),v40,z0,tPen\WObj:=wPaper;
    MoveL Offs(pOrigin,392.90,147.96,0.00),v40,z0,tPen\WObj:=wPaper;
    MoveL Offs(pOrigin,389.45,151.42,0.00),v40,z0,tPen\WObj:=wPaper;
    MoveL Offs(pOrigin,390.05,151.40,0.00),v40,z0,tPen\WObj:=wPaper;
    MoveL Offs(pOrigin,391.86,153.20,0.00),v40,z0,tPen\WObj:=wPaper;
    MoveL Offs(pOrigin,391.52,153.34,0.00),v40,z0,tPen\WObj:=wPaper;
    MoveL Offs(pOrigin,390.46,153.34,0.00),v40,z0,tPen\WObj:=wPaper;
  ENDPROC

  PROC DrawPart140()
    MoveL Offs(pOrigin,389.91,152.75,0.00),v40,z0,tPen\WObj:=wPaper;
    MoveL Offs(pOrigin,391.86,154.70,0.00),v40,z0,tPen\WObj:=wPaper;
    MoveL Offs(pOrigin,392.43,154.40,0.00),v40,z0,tPen\WObj:=wPaper;
    MoveL Offs(pOrigin,388.98,157.86,0.00),v40,z0,tPen\WObj:=wPaper;
    MoveL Offs(pOrigin,389.47,158.29,0.00),v40,z0,tPen\WObj:=wPaper;
    MoveL Offs(pOrigin,391.28,160.09,0.00),v40,z0,tPen\WObj:=wPaper;
    MoveL Offs(pOrigin,390.89,159.67,0.00),v40,z0,tPen\WObj:=wPaper;
    MoveL Offs(pOrigin,389.83,159.67,0.00),v40,z0,tPen\WObj:=wPaper;
    MoveL Offs(pOrigin,389.33,159.64,0.00),v40,z0,tPen\WObj:=wPaper;
    MoveL Offs(pOrigin,391.28,161.59,0.00),v40,z0,tPen\WObj:=wPaper;
    MoveL Offs(pOrigin,391.66,161.15,0.00),v40,z0,tPen\WObj:=wPaper;
    MoveL Offs(pOrigin,388.21,164.60,0.00),v40,z0,tPen\WObj:=wPaper;
    MoveL Offs(pOrigin,388.90,165.18,0.00),v40,z0,tPen\WObj:=wPaper;
    MoveL Offs(pOrigin,390.55,166.83,0.00),v40,z0,tPen\WObj:=wPaper;
    MoveL Offs(pOrigin,390.25,167.06,0.00),v40,z0,tPen\WObj:=wPaper;
    MoveL Offs(pOrigin,389.19,167.06,0.00),v40,z0,tPen\WObj:=wPaper;
    MoveL Offs(pOrigin,388.60,166.38,0.00),v40,z0,tPen\WObj:=wPaper;
    MoveL Offs(pOrigin,390.40,168.18,0.00),v40,z0,tPen\WObj:=wPaper;
    MoveL Offs(pOrigin,391.05,167.74,0.00),v40,z0,tPen\WObj:=wPaper;
    MoveL Offs(pOrigin,387.59,171.19,0.00),v40,z0,tPen\WObj:=wPaper;
    MoveL Offs(pOrigin,388.17,171.92,0.00),v40,z0,tPen\WObj:=wPaper;
    MoveL Offs(pOrigin,389.97,173.72,0.00),v40,z0,tPen\WObj:=wPaper;
    MoveL Offs(pOrigin,389.61,173.40,0.00),v40,z0,tPen\WObj:=wPaper;
    MoveL Offs(pOrigin,388.55,173.40,0.00),v40,z0,tPen\WObj:=wPaper;
    MoveL Offs(pOrigin,388.02,173.26,0.00),v40,z0,tPen\WObj:=wPaper;
    MoveL Offs(pOrigin,389.83,175.07,0.00),v40,z0,tPen\WObj:=wPaper;
    MoveL Offs(pOrigin,389.40,175.51,0.00),v40,z0,tPen\WObj:=wPaper;
    MoveL Offs(pOrigin,388.34,175.51,0.00),v40,z0,tPen\WObj:=wPaper;
    MoveL Offs(pOrigin,387.88,176.11,0.00),v40,z0,tPen\WObj:=wPaper;
    MoveL Offs(pOrigin,389.53,177.76,0.00),v40,z0,tPen\WObj:=wPaper;
    MoveL Offs(pOrigin,390.27,177.48,0.00),v40,z0,tPen\WObj:=wPaper;
    MoveL Offs(pOrigin,386.81,180.93,0.00),v40,z0,tPen\WObj:=wPaper;
    MoveL Offs(pOrigin,387.45,181.65,0.00),v40,z0,tPen\WObj:=wPaper;
    MoveL Offs(pOrigin,389.25,183.45,0.00),v40,z0,tPen\WObj:=wPaper;
    MoveL Offs(pOrigin,389.50,184.22,0.00),v40,z0,tPen\WObj:=wPaper;
    MoveL Offs(pOrigin,386.04,187.68,0.00),v40,z0,tPen\WObj:=wPaper;
    MoveL Offs(pOrigin,386.72,188.39,0.00),v40,z0,tPen\WObj:=wPaper;
    MoveL Offs(pOrigin,388.52,190.19,0.00),v40,z0,tPen\WObj:=wPaper;
    MoveL Offs(pOrigin,388.88,190.81,0.00),v40,z0,tPen\WObj:=wPaper;
    MoveL Offs(pOrigin,385.57,194.12,0.00),v40,z0,tPen\WObj:=wPaper;
    MoveL Offs(pOrigin,385.99,193.63,0.00),v40,z0,tPen\WObj:=wPaper;
    MoveL Offs(pOrigin,387.79,195.43,0.00),v40,z0,tPen\WObj:=wPaper;
    MoveL Offs(pOrigin,388.41,195.76,0.00),v40,z0,tPen\WObj:=wPaper;
    MoveL Offs(pOrigin,385.26,198.91,0.00),v40,z0,tPen\WObj:=wPaper;
    MoveL Offs(pOrigin,385.55,199.17,0.00),v40,z0,tPen\WObj:=wPaper;
    MoveL Offs(pOrigin,387.36,200.97,0.00),v40,z0,tPen\WObj:=wPaper;
    MoveL Offs(pOrigin,387.95,200.70,0.00),v40,z0,tPen\WObj:=wPaper;
    MoveL Offs(pOrigin,384.79,203.86,0.00),v40,z0,tPen\WObj:=wPaper;
    MoveL Offs(pOrigin,385.42,203.52,0.00),v40,z0,tPen\WObj:=wPaper;
    MoveL Offs(pOrigin,387.22,205.32,0.00),v40,z0,tPen\WObj:=wPaper;
    MoveL Offs(pOrigin,387.78,205.35,0.00),v40,z0,tPen\WObj:=wPaper;
    MoveL Offs(pOrigin,384.48,208.65,0.00),v40,z0,tPen\WObj:=wPaper;
    MoveL Offs(pOrigin,384.84,208.91,0.00),v40,z0,tPen\WObj:=wPaper;
    MoveL Offs(pOrigin,386.64,210.71,0.00),v40,z0,tPen\WObj:=wPaper;
    MoveL Offs(pOrigin,387.32,210.29,0.00),v40,z0,tPen\WObj:=wPaper;
    MoveL Offs(pOrigin,384.01,213.60,0.00),v40,z0,tPen\WObj:=wPaper;
    MoveL Offs(pOrigin,384.55,213.10,0.00),v40,z0,tPen\WObj:=wPaper;
    MoveL Offs(pOrigin,386.20,214.75,0.00),v40,z0,tPen\WObj:=wPaper;
    MoveL Offs(pOrigin,386.70,215.39,0.00),v40,z0,tPen\WObj:=wPaper;
    MoveL Offs(pOrigin,379.19,222.90,0.00),v40,z0,tPen\WObj:=wPaper;
    MoveL Offs(pOrigin,379.79,223.27,0.00),v40,z0,tPen\WObj:=wPaper;
    MoveL Offs(pOrigin,381.29,224.77,0.00),v40,fine,tPen\WObj:=wPaper;
    MoveL Offs(pOrigin,381.29,224.77,6.00),v60,z5,tPen\WObj:=wPaper;
    MoveL Offs(pOrigin,382.49,224.48,6.00),vTravel,z5,tPen\WObj:=wPaper;
    MoveL Offs(pOrigin,382.49,224.48,0.00),v60,z0,tPen\WObj:=wPaper;
    MoveL Offs(pOrigin,384.14,226.13,0.00),v40,z0,tPen\WObj:=wPaper;
    MoveL Offs(pOrigin,384.42,226.63,0.00),v40,z0,tPen\WObj:=wPaper;
    MoveL Offs(pOrigin,369.55,241.51,0.00),v40,z0,tPen\WObj:=wPaper;
    MoveL Offs(pOrigin,370.40,240.77,0.00),v40,z0,tPen\WObj:=wPaper;
    MoveL Offs(pOrigin,366.95,237.31,0.00),v40,fine,tPen\WObj:=wPaper;
    MoveL Offs(pOrigin,366.95,237.31,6.00),v60,z5,tPen\WObj:=wPaper;
    MoveL Offs(pOrigin,364.18,234.93,6.00),vTravel,z5,tPen\WObj:=wPaper;
    MoveL Offs(pOrigin,364.18,234.93,0.00),v60,z0,tPen\WObj:=wPaper;
    MoveL Offs(pOrigin,378.30,220.81,0.00),v40,z0,tPen\WObj:=wPaper;
    MoveL Offs(pOrigin,377.68,221.17,0.00),v40,z0,tPen\WObj:=wPaper;
    MoveL Offs(pOrigin,375.58,219.06,0.00),v40,z0,tPen\WObj:=wPaper;
    MoveL Offs(pOrigin,374.56,218.57,0.00),v40,z0,tPen\WObj:=wPaper;
    MoveL Offs(pOrigin,378.32,214.81,0.00),v40,z0,tPen\WObj:=wPaper;
    MoveL Offs(pOrigin,377.97,215.48,0.00),v40,z0,tPen\WObj:=wPaper;
    MoveL Offs(pOrigin,375.56,213.07,0.00),v40,z0,tPen\WObj:=wPaper;
    MoveL Offs(pOrigin,376.22,213.53,0.00),v40,z0,tPen\WObj:=wPaper;
    MoveL Offs(pOrigin,377.29,213.53,0.00),v40,z0,tPen\WObj:=wPaper;
    MoveL Offs(pOrigin,378.17,213.47,0.00),v40,z0,tPen\WObj:=wPaper;
    MoveL Offs(pOrigin,374.57,217.07,0.00),v40,z0,tPen\WObj:=wPaper;
    MoveL Offs(pOrigin,375.27,217.27,0.00),v40,z0,tPen\WObj:=wPaper;
    MoveL Offs(pOrigin,377.98,219.97,0.00),v40,z0,tPen\WObj:=wPaper;
    MoveL Offs(pOrigin,378.60,219.01,0.00),v40,z0,tPen\WObj:=wPaper;
    MoveL Offs(pOrigin,372.14,225.47,0.00),v40,fine,tPen\WObj:=wPaper;
    MoveL Offs(pOrigin,372.14,225.47,6.00),v60,z5,tPen\WObj:=wPaper;
    MoveL Offs(pOrigin,371.98,227.27,6.00),vTravel,z5,tPen\WObj:=wPaper;
    MoveL Offs(pOrigin,371.98,227.27,0.00),v60,z0,tPen\WObj:=wPaper;
    MoveL Offs(pOrigin,371.55,227.91,0.00),v40,z0,tPen\WObj:=wPaper;
    MoveL Offs(pOrigin,371.98,227.27,0.00),v40,z0,tPen\WObj:=wPaper;
    MoveL Offs(pOrigin,372.43,228.16,0.00),v40,z0,tPen\WObj:=wPaper;
    MoveL Offs(pOrigin,367.33,233.27,0.00),v40,fine,tPen\WObj:=wPaper;
    MoveL Offs(pOrigin,367.33,233.27,6.00),v60,z5,tPen\WObj:=wPaper;
    MoveL Offs(pOrigin,365.53,232.08,6.00),vTravel,z5,tPen\WObj:=wPaper;
    MoveL Offs(pOrigin,365.53,232.08,0.00),v60,z0,tPen\WObj:=wPaper;
    MoveL Offs(pOrigin,362.08,235.54,0.00),v40,z0,tPen\WObj:=wPaper;
    MoveL Offs(pOrigin,361.70,235.05,0.00),v40,z0,tPen\WObj:=wPaper;
    MoveL Offs(pOrigin,360.95,234.30,0.00),v40,z0,tPen\WObj:=wPaper;
    MoveL Offs(pOrigin,361.03,233.59,0.00),v40,z0,tPen\WObj:=wPaper;
    MoveL Offs(pOrigin,358.03,236.60,0.00),v40,z0,tPen\WObj:=wPaper;
    MoveL Offs(pOrigin,358.25,236.09,0.00),v40,z0,tPen\WObj:=wPaper;
    MoveL Offs(pOrigin,357.35,235.19,0.00),v40,z0,tPen\WObj:=wPaper;
    MoveL Offs(pOrigin,358.40,234.74,0.00),v40,z0,tPen\WObj:=wPaper;
    MoveL Offs(pOrigin,359.45,235.79,0.00),v40,fine,tPen\WObj:=wPaper;
    MoveL Offs(pOrigin,359.45,235.79,6.00),v60,z5,tPen\WObj:=wPaper;
    MoveL Offs(pOrigin,359.75,234.59,6.00),vTravel,z5,tPen\WObj:=wPaper;
    MoveL Offs(pOrigin,359.75,234.59,0.00),v60,z0,tPen\WObj:=wPaper;
    MoveL Offs(pOrigin,360.65,235.50,0.00),v40,fine,tPen\WObj:=wPaper;
    MoveL Offs(pOrigin,360.65,235.50,6.00),v60,z5,tPen\WObj:=wPaper;
    MoveL Offs(pOrigin,359.08,234.05,6.00),vTravel,z5,tPen\WObj:=wPaper;
    MoveL Offs(pOrigin,359.08,234.05,0.00),v60,z0,tPen\WObj:=wPaper;
    MoveL Offs(pOrigin,356.08,237.05,0.00),v40,z0,tPen\WObj:=wPaper;
    MoveL Offs(pOrigin,355.71,236.53,0.00),v40,z0,tPen\WObj:=wPaper;
    MoveL Offs(pOrigin,354.81,235.63,0.00),v40,z0,tPen\WObj:=wPaper;
    MoveL Offs(pOrigin,354.36,236.68,0.00),v40,z0,tPen\WObj:=wPaper;
    MoveL Offs(pOrigin,353.46,235.77,0.00),v40,z0,tPen\WObj:=wPaper;
    MoveL Offs(pOrigin,353.84,234.81,0.00),v40,z0,tPen\WObj:=wPaper;
  ENDPROC

  PROC DrawPart141()
    MoveL Offs(pOrigin,350.83,237.82,0.00),v40,z0,tPen\WObj:=wPaper;
    MoveL Offs(pOrigin,350.62,237.41,0.00),v40,z0,tPen\WObj:=wPaper;
    MoveL Offs(pOrigin,349.42,236.21,0.00),v40,z0,tPen\WObj:=wPaper;
    MoveL Offs(pOrigin,348.59,235.58,0.00),v40,z0,tPen\WObj:=wPaper;
    MoveL Offs(pOrigin,345.74,238.43,0.00),v40,z0,tPen\WObj:=wPaper;
    MoveL Offs(pOrigin,345.38,238.15,0.00),v40,z0,tPen\WObj:=wPaper;
    MoveL Offs(pOrigin,344.03,236.79,0.00),v40,z0,tPen\WObj:=wPaper;
    MoveL Offs(pOrigin,343.65,236.04,0.00),v40,z0,tPen\WObj:=wPaper;
    MoveL Offs(pOrigin,340.64,239.05,0.00),v40,z0,tPen\WObj:=wPaper;
    MoveL Offs(pOrigin,341.34,238.58,0.00),v40,z0,tPen\WObj:=wPaper;
    MoveL Offs(pOrigin,339.98,237.23,0.00),v40,z0,tPen\WObj:=wPaper;
    MoveL Offs(pOrigin,340.20,236.50,0.00),v40,z0,tPen\WObj:=wPaper;
    MoveL Offs(pOrigin,337.35,239.36,0.00),v40,z0,tPen\WObj:=wPaper;
    MoveL Offs(pOrigin,337.29,239.02,0.00),v40,z0,tPen\WObj:=wPaper;
    MoveL Offs(pOrigin,335.94,237.67,0.00),v40,z0,tPen\WObj:=wPaper;
    MoveL Offs(pOrigin,335.26,236.97,0.00),v40,z0,tPen\WObj:=wPaper;
    MoveL Offs(pOrigin,332.40,239.82,0.00),v40,z0,tPen\WObj:=wPaper;
    MoveL Offs(pOrigin,331.90,239.60,0.00),v40,z0,tPen\WObj:=wPaper;
    MoveL Offs(pOrigin,330.55,238.25,0.00),v40,z0,tPen\WObj:=wPaper;
    MoveL Offs(pOrigin,330.31,237.43,0.00),v40,z0,tPen\WObj:=wPaper;
    MoveL Offs(pOrigin,327.61,240.14,0.00),v40,z0,tPen\WObj:=wPaper;
    MoveL Offs(pOrigin,327.56,239.74,0.00),v40,z0,tPen\WObj:=wPaper;
    MoveL Offs(pOrigin,326.20,238.39,0.00),v40,z0,tPen\WObj:=wPaper;
    MoveL Offs(pOrigin,325.52,237.75,0.00),v40,z0,tPen\WObj:=wPaper;
    MoveL Offs(pOrigin,322.66,240.60,0.00),v40,z0,tPen\WObj:=wPaper;
    MoveL Offs(pOrigin,322.02,240.17,0.00),v40,z0,tPen\WObj:=wPaper;
    MoveL Offs(pOrigin,320.66,238.82,0.00),v40,z0,tPen\WObj:=wPaper;
    MoveL Offs(pOrigin,320.72,238.06,0.00),v40,z0,tPen\WObj:=wPaper;
    MoveL Offs(pOrigin,318.17,240.61,0.00),v40,z0,tPen\WObj:=wPaper;
    MoveL Offs(pOrigin,317.67,240.31,0.00),v40,z0,tPen\WObj:=wPaper;
    MoveL Offs(pOrigin,316.32,238.96,0.00),v40,z0,tPen\WObj:=wPaper;
    MoveL Offs(pOrigin,316.08,238.22,0.00),v40,z0,tPen\WObj:=wPaper;
    MoveL Offs(pOrigin,313.37,240.93,0.00),v40,z0,tPen\WObj:=wPaper;
    MoveL Offs(pOrigin,313.18,240.29,0.00),v40,z0,tPen\WObj:=wPaper;
    MoveL Offs(pOrigin,311.98,239.09,0.00),v40,z0,tPen\WObj:=wPaper;
    MoveL Offs(pOrigin,311.28,238.54,0.00),v40,z0,tPen\WObj:=wPaper;
    MoveL Offs(pOrigin,308.88,240.94,0.00),v40,z0,tPen\WObj:=wPaper;
    MoveL Offs(pOrigin,308.68,240.28,0.00),v40,z0,tPen\WObj:=wPaper;
    MoveL Offs(pOrigin,307.63,239.23,0.00),v40,z0,tPen\WObj:=wPaper;
    MoveL Offs(pOrigin,308.29,238.55,0.00),v40,z0,tPen\WObj:=wPaper;
    MoveL Offs(pOrigin,305.73,241.10,0.00),v40,z0,tPen\WObj:=wPaper;
    MoveL Offs(pOrigin,305.69,240.27,0.00),v40,z0,tPen\WObj:=wPaper;
    MoveL Offs(pOrigin,304.79,239.37,0.00),v40,z0,tPen\WObj:=wPaper;
    MoveL Offs(pOrigin,305.29,238.56,0.00),v40,z0,tPen\WObj:=wPaper;
    MoveL Offs(pOrigin,302.89,240.96,0.00),v40,z0,tPen\WObj:=wPaper;
    MoveL Offs(pOrigin,302.69,240.26,0.00),v40,z0,tPen\WObj:=wPaper;
    MoveL Offs(pOrigin,301.79,239.36,0.00),v40,z0,tPen\WObj:=wPaper;
    MoveL Offs(pOrigin,302.30,238.57,0.00),v40,z0,tPen\WObj:=wPaper;
    MoveL Offs(pOrigin,300.04,240.82,0.00),v40,z0,tPen\WObj:=wPaper;
    MoveL Offs(pOrigin,299.55,240.10,0.00),v40,z0,tPen\WObj:=wPaper;
    MoveL Offs(pOrigin,298.79,239.35,0.00),v40,z0,tPen\WObj:=wPaper;
    MoveL Offs(pOrigin,299.30,238.58,0.00),v40,z0,tPen\WObj:=wPaper;
    MoveL Offs(pOrigin,296.00,241.88,0.00),v40,z0,tPen\WObj:=wPaper;
    MoveL Offs(pOrigin,296.55,241.59,0.00),v40,z0,tPen\WObj:=wPaper;
    MoveL Offs(pOrigin,301.66,246.70,0.00),v40,fine,tPen\WObj:=wPaper;
    MoveL Offs(pOrigin,301.66,246.70,6.00),v60,z5,tPen\WObj:=wPaper;
    MoveL Offs(pOrigin,300.32,246.85,6.00),vTravel,z5,tPen\WObj:=wPaper;
    MoveL Offs(pOrigin,300.32,246.85,0.00),v60,z0,tPen\WObj:=wPaper;
    MoveL Offs(pOrigin,297.16,243.69,0.00),v40,z0,tPen\WObj:=wPaper;
    MoveL Offs(pOrigin,296.59,244.28,0.00),v40,z0,tPen\WObj:=wPaper;
    MoveL Offs(pOrigin,299.14,241.72,0.00),v40,z0,tPen\WObj:=wPaper;
    MoveL Offs(pOrigin,298.65,242.20,0.00),v40,z0,tPen\WObj:=wPaper;
    MoveL Offs(pOrigin,293.69,237.24,0.00),v40,z0,tPen\WObj:=wPaper;
    MoveL Offs(pOrigin,293.76,236.65,0.00),v40,z0,tPen\WObj:=wPaper;
    MoveL Offs(pOrigin,290.01,240.40,0.00),v40,z0,tPen\WObj:=wPaper;
    MoveL Offs(pOrigin,290.56,240.08,0.00),v40,z0,tPen\WObj:=wPaper;
    MoveL Offs(pOrigin,291.91,241.43,0.00),v40,z0,tPen\WObj:=wPaper;
    MoveL Offs(pOrigin,292.55,240.84,0.00),v40,z0,tPen\WObj:=wPaper;
    MoveL Offs(pOrigin,290.00,243.40,0.00),v40,z0,tPen\WObj:=wPaper;
    MoveL Offs(pOrigin,291.01,243.85,0.00),v40,z0,tPen\WObj:=wPaper;
    MoveL Offs(pOrigin,291.58,243.43,0.00),v40,z0,tPen\WObj:=wPaper;
    MoveL Offs(pOrigin,291.86,240.45,0.00),v40,z0,tPen\WObj:=wPaper;
    MoveL Offs(pOrigin,292.71,239.10,0.00),v40,z0,tPen\WObj:=wPaper;
    MoveL Offs(pOrigin,293.99,238.75,0.00),v40,z0,tPen\WObj:=wPaper;
    MoveL Offs(pOrigin,295.05,239.10,0.00),v40,z0,tPen\WObj:=wPaper;
    MoveL Offs(pOrigin,296.68,240.88,0.00),v40,z0,tPen\WObj:=wPaper;
    MoveL Offs(pOrigin,298.66,250.44,0.00),v40,z0,tPen\WObj:=wPaper;
    MoveL Offs(pOrigin,302.06,264.04,0.00),v40,z0,tPen\WObj:=wPaper;
    MoveL Offs(pOrigin,301.85,266.38,0.00),v40,z0,tPen\WObj:=wPaper;
    MoveL Offs(pOrigin,301.07,269.14,0.00),v40,z0,tPen\WObj:=wPaper;
    MoveL Offs(pOrigin,299.80,271.90,0.00),v40,z0,tPen\WObj:=wPaper;
    MoveL Offs(pOrigin,298.45,273.39,0.00),v40,z0,tPen\WObj:=wPaper;
    MoveL Offs(pOrigin,296.33,274.24,0.00),v40,z0,tPen\WObj:=wPaper;
    MoveL Offs(pOrigin,294.84,274.02,0.00),v40,z0,tPen\WObj:=wPaper;
    MoveL Offs(pOrigin,293.56,273.46,0.00),v40,z0,tPen\WObj:=wPaper;
    MoveL Offs(pOrigin,291.44,271.48,0.00),v40,z0,tPen\WObj:=wPaper;
    MoveL Offs(pOrigin,291.44,271.48,0.00),v40,z0,tPen\WObj:=wPaper;
    MoveL Offs(pOrigin,291.44,270.41,0.00),v40,z0,tPen\WObj:=wPaper;
    MoveL Offs(pOrigin,290.38,269.99,0.00),v40,z0,tPen\WObj:=wPaper;
    MoveL Offs(pOrigin,290.38,269.99,0.00),v40,z0,tPen\WObj:=wPaper;
    MoveL Offs(pOrigin,290.16,270.41,0.00),v40,z0,tPen\WObj:=wPaper;
    MoveL Offs(pOrigin,290.38,271.05,0.00),v40,z0,tPen\WObj:=wPaper;
    MoveL Offs(pOrigin,291.44,271.48,0.00),v40,z0,tPen\WObj:=wPaper;
    MoveL Offs(pOrigin,290.41,271.47,0.00),v40,z0,tPen\WObj:=wPaper;
    MoveL Offs(pOrigin,290.41,273.60,0.00),v40,fine,tPen\WObj:=wPaper;
    MoveL Offs(pOrigin,290.41,273.60,6.00),v60,z5,tPen\WObj:=wPaper;
    MoveL Offs(pOrigin,292.53,273.60,6.00),vTravel,z5,tPen\WObj:=wPaper;
    MoveL Offs(pOrigin,292.53,273.60,0.00),v60,z0,tPen\WObj:=wPaper;
    MoveL Offs(pOrigin,292.53,277.21,0.00),v40,z0,tPen\WObj:=wPaper;
    MoveL Offs(pOrigin,292.50,277.94,0.00),v40,z0,tPen\WObj:=wPaper;
    MoveL Offs(pOrigin,299.09,277.94,0.00),v40,z0,tPen\WObj:=wPaper;
    MoveL Offs(pOrigin,299.30,276.89,0.00),v40,z0,tPen\WObj:=wPaper;
    MoveL Offs(pOrigin,288.46,276.89,0.00),v40,z0,tPen\WObj:=wPaper;
    MoveL Offs(pOrigin,287.83,277.00,0.00),v40,z0,tPen\WObj:=wPaper;
    MoveL Offs(pOrigin,288.04,277.78,0.00),v40,z0,tPen\WObj:=wPaper;
    MoveL Offs(pOrigin,289.24,277.92,0.00),v40,z0,tPen\WObj:=wPaper;
    MoveL Offs(pOrigin,289.31,278.49,0.00),v40,fine,tPen\WObj:=wPaper;
    MoveL Offs(pOrigin,289.31,278.49,6.00),v60,z5,tPen\WObj:=wPaper;
    MoveL Offs(pOrigin,289.95,276.58,6.00),vTravel,z5,tPen\WObj:=wPaper;
    MoveL Offs(pOrigin,289.95,276.58,0.00),v60,z0,tPen\WObj:=wPaper;
    MoveL Offs(pOrigin,288.25,276.58,0.00),v40,z0,tPen\WObj:=wPaper;
    MoveL Offs(pOrigin,287.83,277.00,0.00),v40,z0,tPen\WObj:=wPaper;
    MoveL Offs(pOrigin,287.83,277.00,0.00),v40,z0,tPen\WObj:=wPaper;
    MoveL Offs(pOrigin,286.12,276.72,0.00),v40,z0,tPen\WObj:=wPaper;
    MoveL Offs(pOrigin,286.55,275.73,0.00),v40,z0,tPen\WObj:=wPaper;
    MoveL Offs(pOrigin,287.25,275.94,0.00),v40,z0,tPen\WObj:=wPaper;
    MoveL Offs(pOrigin,287.25,274.66,0.00),v40,z0,tPen\WObj:=wPaper;
    MoveL Offs(pOrigin,288.30,274.66,0.00),v40,z0,tPen\WObj:=wPaper;
    MoveL Offs(pOrigin,288.30,275.94,0.00),v40,fine,tPen\WObj:=wPaper;
    MoveL Offs(pOrigin,288.30,275.94,6.00),v60,z5,tPen\WObj:=wPaper;
  ENDPROC

